FUNCTION "HMI animation unit" : VOID	// FC 60
TITLE = HMI ANIMATION FUNCTION
AUTHOR : Milesi
VERSION : 0.1
VAR_TEMP
  Temp_Start : BOOL ;
  Temp_Alm : BOOL ;
  Temp_Aux : BOOL ;
END_VAR
BEGIN
NETWORK
TITLE = LINE
      AN    "M197.0";
      =     "HMI animation".Line.DB60_DBX156_0;
NETWORK
TITLE = ALARMS PRESENT TO HMI 
      AN    "M102.1";
      O     "Db Plc <=> HMI".LINE1.DB100_DBX149_7;
      =     "HMI animation".Line.DB60_DBX156_1;
NETWORK
TITLE = LINE RUN WITH ZERO SPEED
      A     "M180.1";
      =     "HMI animation".Line.DB60_DBX156_2;
NETWORK
TITLE = PLC <--> HMI COMUNICATION CONTROL
      AN    "HMI animation".Line.DB60_DBX156_7;
      S     "HMI animation".Line.DB60_DBX156_7;
NETWORK
TITLE = TAKE-UP UNIT
// General alarm
      A(;
      ON    "M195.0";
      ON    "M195.1";
      O     "Db Plc <=> HMI".TAKE_UP_1.DB100_DBX107_2;
      );
      =     "HMI animation".Take_up_unit.DB60_DBX0_0;
// Driven pintle emergency
      A     "Db Plc <=> HMI".TRAVERSE.DB100_DBX105_0;
      =     "HMI animation".Take_up_unit.DB60_DBX0_1;
// Idle pintle emergency
      A     "Db Plc <=> HMI".TRAVERSE.DB100_DBX105_1;
      =     "HMI animation".Take_up_unit.DB60_DBX0_2;
// Bobbin up-down
      A     "MAP_DI".DB91_DBX006_0;
      A     "MAP_DI".DB91_DBX006_2;
      =     "HMI animation".Take_up_unit.DB60_DBX0_3;
// Traverse right direction
      AN    "M10.1";
      =     "HMI animation".Take_up_unit.DB60_DBX0_4;
// Traverse left direction
      A     "M10.1";
      =     "HMI animation".Take_up_unit.DB60_DBX0_5;
// Bobbin motor status
      A     "Db Plc <=> HMI".TAKE_UP_1.DB100_DBX107_4;
      O     "Db Plc <=> HMI".TAKE_UP_1.DB100_DBX107_5;
      O     "Db Plc <=> HMI".TAKE_UP_1.DB100_DBX107_6;
      =     #Temp_Aux;
      CALL  "Motor status HMI" (
           Start                    := "Plc --> Drives".BOBBIN_CONTROL_W1.DB2_DBX41_0,
           Fault                    := #Temp_Aux,
           Status_Reg               := "HMI animation".Take_up_unit.DB60_DBB1);
// Bobbin blower status
      CALL  "Motor status HMI" (
           Start                    := "MAP_DO".DB93_DBX005_1,
           Fault                    := "Db Plc <=> HMI".TAKE_UP_1.DB100_DBX107_3,
           Status_Reg               := "HMI animation".Take_up_unit.DB60_DBB2);
// Traverse motor status
      CALL  "Motor status HMI" (
           Start                    := "Plc --> Drives".TRAVERSE_CONTROL_W1.DB2_DBX1_0,
           Fault                    := "Db Plc <=> HMI".TRAVERSE.DB100_DBX105_3,
           Status_Reg               := "HMI animation".Take_up_unit.DB60_DBB3);
// Traverse blower status
      CALL  "Motor status HMI" (
           Start                    := "MAP_DO".DB93_DBX005_0,
           Fault                    := "Db Plc <=> HMI".TRAVERSE.DB100_DBX105_2,
           Status_Reg               := "HMI animation".Take_up_unit.DB60_DBB4);
// Bobbin driven pintle motor status
      A     "MAP_DO".DB93_DBX004_2;
      O     "MAP_DO".DB93_DBX004_3;
      =     #Temp_Start;
      CALL  "Motor status HMI" (
           Start                    := #Temp_Start,
           Fault                    := "Db Plc <=> HMI".TAKE_UP_1.DB100_DBX107_2,
           Status_Reg               := "HMI animation".Take_up_unit.DB60_DBB5);
// Bobbin idle pintle motor status
      A     "MAP_DO".DB93_DBX004_0;
      O     "MAP_DO".DB93_DBX004_1;
      =     #Temp_Start;
      CALL  "Motor status HMI" (
           Start                    := #Temp_Start,
           Fault                    := "Db Plc <=> HMI".TAKE_UP_1.DB100_DBX107_2,
           Status_Reg               := "HMI animation".Take_up_unit.DB60_DBB6);
// Bobbin pintle opening-closing motor status
      A     "MAP_DO".DB93_DBX004_4;
      O     "MAP_DO".DB93_DBX004_5;
      =     #Temp_Start;
      CALL  "Motor status HMI" (
           Start                    := #Temp_Start,
           Fault                    := "Db Plc <=> HMI".TAKE_UP_1.DB100_DBX107_2,
           Status_Reg               := "HMI animation".Take_up_unit.DB60_DBB7);
NETWORK
TITLE = CAPSTAN
// General alarm
      AN    "M197.3";
      =     "HMI animation".Capstan.DB60_DBX12_0;
// Cable block
      A     "MAP_DI".DB91_DBX012_3;
      =     "HMI animation".Capstan.DB60_DBX12_1;
// Motor status
      A     "Db Plc <=> HMI".CAPSTAN.DB100_DBX109_6;
      O     "Db Plc <=> HMI".CAPSTAN.DB100_DBX109_7;
      =     #Temp_Alm;
      CALL  "Motor status HMI" (
           Start                    := "Plc --> Drives".CAPSTAN_CONTROL_W1.DB2_DBX81_0,
           Fault                    := #Temp_Alm,
           Status_Reg               := "HMI animation".Capstan.DB60_DBB13);
// Blower status
      CALL  "Motor status HMI" (
           Start                    := "MAP_DO".DB93_DBX001_2,
           Fault                    := "Db Plc <=> HMI".CAPSTAN.DB100_DBX109_0,
           Status_Reg               := "HMI animation".Capstan.DB60_DBB14);
NETWORK
TITLE = CAGE 24
// General alarm
      AN    "M195.3";
      O     "Db Plc <=> HMI".CAGE24_1.DB100_DBX112_02;
      O     "Db Plc <=> HMI".CAGE24_1.DB100_DBX112_04;
      O     "Db Plc <=> HMI".CAGE24_1.DB100_DBX113_05;
      =     "HMI animation".Cage_24.DB60_DBX36_0;
// Motor status
      A     "Db Plc <=> HMI".CAGE24_4.DB100_DBX118_05;
      O     "Db Plc <=> HMI".CAGE24_4.DB100_DBX118_06;
      =     #Temp_Alm;
      CALL  "Motor status HMI" (
           Start                    := "Plc --> Drives".CAGE_24_CONTROL_W1.DB2_DBX161_0,
           Fault                    := #Temp_Alm,
           Status_Reg               := "HMI animation".Cage_24.DB60_DBB37);
// Blower status
      CALL  "Motor status HMI" (
           Start                    := "MAP_DO".DB93_DBX018_2,
           Fault                    := "Db Plc <=> HMI".CAGE24_1.DB100_DBX113_02,
           Status_Reg               := "HMI animation".Cage_24.DB60_DBB38);
// Loading motor status
      A     "MAP_DO".DB93_DBX018_4;
      O     "MAP_DO".DB93_DBX018_3;
      =     #Temp_Start;
      CALL  "Motor status HMI" (
           Start                    := #Temp_Start,
           Fault                    := "Db Plc <=> HMI".CAGE24_1.DB100_DBX112_04,
           Status_Reg               := "HMI animation".Cage_24.DB60_DBB39);
NETWORK
TITLE = CAGE 24 PREFORMING
// General alarm
      AN    "M195.4";
      =     "HMI animation".Cage_24_preforming.DB60_DBX48_0;
// Motor status
      A     "Db Plc <=> HMI".CAGE24_4.DB100_DBX119_04;
      O     "Db Plc <=> HMI".CAGE24_4.DB100_DBX119_07;
      =     #Temp_Alm;
      CALL  "Motor status HMI" (
           Start                    := "Plc --> Drives".CAGE_24_PREF_CONTROL_W1.DB2_DBX121_0,
           Fault                    := #Temp_Alm,
           Status_Reg               := "HMI animation".Cage_24_preforming.DB60_DBB49);
// Blower status
      CALL  "Motor status HMI" (
           Start                    := "MAP_DO".DB93_DBX018_1,
           Fault                    := "Db Plc <=> HMI".CAGE24_4.DB100_DBX119_05,
           Status_Reg               := "HMI animation".Cage_24_preforming.DB60_DBB50);
NETWORK
TITLE = CAGE 18
// General alarm
      AN    "M195.5";
      O     "Db Plc <=> HMI".CAGE18_1.DB100_DBX120_02;
      O     "Db Plc <=> HMI".CAGE18_1.DB100_DBX120_04;
      O     "Db Plc <=> HMI".CAGE18_1.DB100_DBX121_05;
      =     "HMI animation".Cage_18.DB60_DBX60_0;
// Motor status
      A     "Db Plc <=> HMI".CAGE18_4.DB100_DBX126_05;
      O     "Db Plc <=> HMI".CAGE18_4.DB100_DBX126_06;
      =     #Temp_Alm;
      CALL  "Motor status HMI" (
           Start                    := "Plc --> Drives".CAGE_18_CONTROL_W1.DB2_DBX241_0,
           Fault                    := #Temp_Alm,
           Status_Reg               := "HMI animation".Cage_18.DB60_DBB61);
// Blower status
      CALL  "Motor status HMI" (
           Start                    := "MAP_DO".DB93_DBX028_2,
           Fault                    := "Db Plc <=> HMI".CAGE18_1.DB100_DBX121_02,
           Status_Reg               := "HMI animation".Cage_18.DB60_DBB62);
// Loading motor status
      A     "MAP_DO".DB93_DBX028_4;
      O     "MAP_DO".DB93_DBX028_3;
      =     #Temp_Start;
      CALL  "Motor status HMI" (
           Start                    := #Temp_Start,
           Fault                    := "Db Plc <=> HMI".CAGE18_1.DB100_DBX120_04,
           Status_Reg               := "HMI animation".Cage_18.DB60_DBB63);
NETWORK
TITLE = CAGE 18 PREFORMING
// General alarm
      AN    "M195.6";
      =     "HMI animation".Cage_18_preforming.DB60_DBX72_0;
// Motor status
      A     "Db Plc <=> HMI".CAGE18_4.DB100_DBX127_04;
      O     "Db Plc <=> HMI".CAGE18_4.DB100_DBX127_07;
      =     #Temp_Alm;
      CALL  "Motor status HMI" (
           Start                    := "Plc --> Drives".CAGE_18_PREF_CONTROL_W1.DB2_DBX201_0,
           Fault                    := #Temp_Alm,
           Status_Reg               := "HMI animation".Cage_18_preforming.DB60_DBB73);
// Blower status
      CALL  "Motor status HMI" (
           Start                    := "MAP_DO".DB93_DBX028_1,
           Fault                    := "Db Plc <=> HMI".CAGE18_4.DB100_DBX127_05,
           Status_Reg               := "HMI animation".Cage_18_preforming.DB60_DBB74);
NETWORK
TITLE = CAGE 12
// General alarm
      AN    "M195.7";
      O     "Db Plc <=> HMI".CAGE12_1.DB100_DBX128_02;
      O     "Db Plc <=> HMI".CAGE12_1.DB100_DBX128_06;
      O     "Db Plc <=> HMI".CAGE12_1.DB100_DBX129_05;
      =     "HMI animation".Cage_12.DB60_DBX84_0;
// Motor status
      A     "Db Plc <=> HMI".Cage12_4.DB100_DBX134_05;
      O     "Db Plc <=> HMI".Cage12_4.DB100_DBX134_06;
      =     #Temp_Alm;
      CALL  "Motor status HMI" (
           Start                    := "Plc --> Drives".CAGE_12_CONTROL_W1.DB2_DBX321_0,
           Fault                    := #Temp_Alm,
           Status_Reg               := "HMI animation".Cage_12.DB60_DBB85);
// Blower status
      CALL  "Motor status HMI" (
           Start                    := "MAP_DO".DB93_DBX038_2,
           Fault                    := "Db Plc <=> HMI".CAGE12_1.DB100_DBX129_02,
           Status_Reg               := "HMI animation".Cage_12.DB60_DBB86);
// Loading motor status
      A     "MAP_DO".DB93_DBX038_4;
      O     "MAP_DO".DB93_DBX038_3;
      =     #Temp_Start;
      CALL  "Motor status HMI" (
           Start                    := #Temp_Start,
           Fault                    := "Db Plc <=> HMI".CAGE12_1.DB100_DBX128_06,
           Status_Reg               := "HMI animation".Cage_12.DB60_DBB87);
NETWORK
TITLE = CAGE 12 PREFORMING
// General alarm
      AN    "M196.0";
      =     "HMI animation".Cage_12_preforming.DB60_DBX96_0;
// Motor status
      A     "Db Plc <=> HMI".Cage12_4.DB100_DBX135_04;
      O     "Db Plc <=> HMI".Cage12_4.DB100_DBX135_07;
      =     #Temp_Alm;
      CALL  "Motor status HMI" (
           Start                    := "Plc --> Drives".CAGE_12_PREF_CONTROL_W1.DB2_DBX281_0,
           Fault                    := #Temp_Alm,
           Status_Reg               := "HMI animation".Cage_12_preforming.DB60_DBB97);
// Blower status
      CALL  "Motor status HMI" (
           Start                    := "MAP_DO".DB93_DBX038_1,
           Fault                    := "Db Plc <=> HMI".Cage12_4.DB100_DBX135_05,
           Status_Reg               := "HMI animation".Cage_12_preforming.DB60_DBB98);
NETWORK
TITLE = CAGE 6
// General alarm
      AN    "M196.1";
      O     "Db Plc <=> HMI".Cage6_1.DB100_DBX136_2;
      O     "Db Plc <=> HMI".Cage6_1.DB100_DBX136_6;
      O     "Db Plc <=> HMI".Cage6_1.DB100_DBX137_5;
      =     "HMI animation".Cage_6.DB60_DBX108_0;
// Motor status
      A     "Db Plc <=> HMI".Cage6_4.DB100_DBX142_5;
      O     "Db Plc <=> HMI".Cage6_4.DB100_DBX142_6;
      =     #Temp_Alm;
      CALL  "Motor status HMI" (
           Start                    := "Plc --> Drives".CAGE_6_CONTROL_W1.DB2_DBX361_0,
           Fault                    := #Temp_Alm,
           Status_Reg               := "HMI animation".Cage_6.DB60_DBB109);
// Blower status
      CALL  "Motor status HMI" (
           Start                    := "MAP_DO".DB93_DBX048_2,
           Fault                    := "Db Plc <=> HMI".Cage6_1.DB100_DBX137_2,
           Status_Reg               := "HMI animation".Cage_6.DB60_DBB110);
// Loading motor status
      A     "MAP_DO".DB93_DBX048_3;
      O     "MAP_DO".DB93_DBX048_4;
      =     #Temp_Start;
      CALL  "Motor status HMI" (
           Start                    := #Temp_Start,
           Fault                    := "Db Plc <=> HMI".Cage6_1.DB100_DBX136_6,
           Status_Reg               := "HMI animation".Cage_6.DB60_DBB111);
NETWORK
TITLE = CAGE 6 PREFORMING
// General alarm
      AN    "M196.2";
      =     "HMI animation".Cage_6_preforming.DB60_DBX120_0;
NETWORK
TITLE = PAY-OFF 630 UNIT
// General alarm
      AN    "M196.3";
      =     "HMI animation".Pay_off_630.DB60_DBX132_0;
      A     "MAP_DI".DB91_DBX099_0;
      =     "HMI animation".Pay_off_630.DB60_DBX132_1;
END_FUNCTION

FUNCTION "Take-up traverse impulse" : VOID	// FC 61
TITLE = TAKE-UP TRAVERSE IMPULSES FUNCTION
AUTHOR : Milesi
VERSION : 0.1
VAR_TEMP
  Traverse_Encoder_Caunt : DINT ;
END_VAR
BEGIN
NETWORK
TITLE = COUNT 24V/100kHz SETTINGS
//Presettings
      L     0;
      T     "Count setting".DINT0;
      T     "Count setting".DINT4;
      SET;
      S     DB101.DBX 4.0;
//Command interface writing
      L     "Count setting".DINT0;
      T     "PAD272";
      L     DB101.DBW 4;
      T     "PAW276";
//Status interface reading
      L     "PED272";
      T     "Count setting".DINT8;
      L     "PED276";
      T     "Count setting".DINT12;
NETWORK
TITLE = TAKE-UP TRAVERSE ENCODER COUNT
      L     "Count setting".DINT8;
      NEGD;
      T     #Traverse_Encoder_Caunt;
NETWORK
TITLE = TAKE-UP TRAVERSE POSITION QUOTA CALCULATION
      L     #Traverse_Encoder_Caunt;
      L     "Take-up traverse".DB5_DBD44;
      -D;
      DTR;
      L     1.793919e-03;
      *R;
      T     "Take-up traverse".DB5_DBD40;
      L     #Traverse_Encoder_Caunt;
      T     "Take-up traverse".DB5_DBD44;
NETWORK
TITLE = TRAVERSE QUOTA INCREASE
      L     "Take-up traverse".DB5_DBD40;
      L     "Take-up traverse".DB5_DBD32;
      +R;
      T     "Take-up traverse".DB5_DBD32;
NETWORK
TITLE = TAKE-UP TRAVERSE POSITION QUOTA RESET
      A     "MAP_DI".DB91_DBX008_4;
      JNB   _023;
      L     0.000000e+00;
      T     "Take-up traverse".DB5_DBD32;
_023: NOP   0;
END_FUNCTION

FUNCTION "Cage 24 wires insertion" : VOID	// FC 70
TITLE = CAGE 24 WIRES INSERTION AND ALARM FUNCTION
AUTHOR : Milesi
VERSION : 0.1
VAR_TEMP
  Tres : BOOL ;
END_VAR
BEGIN
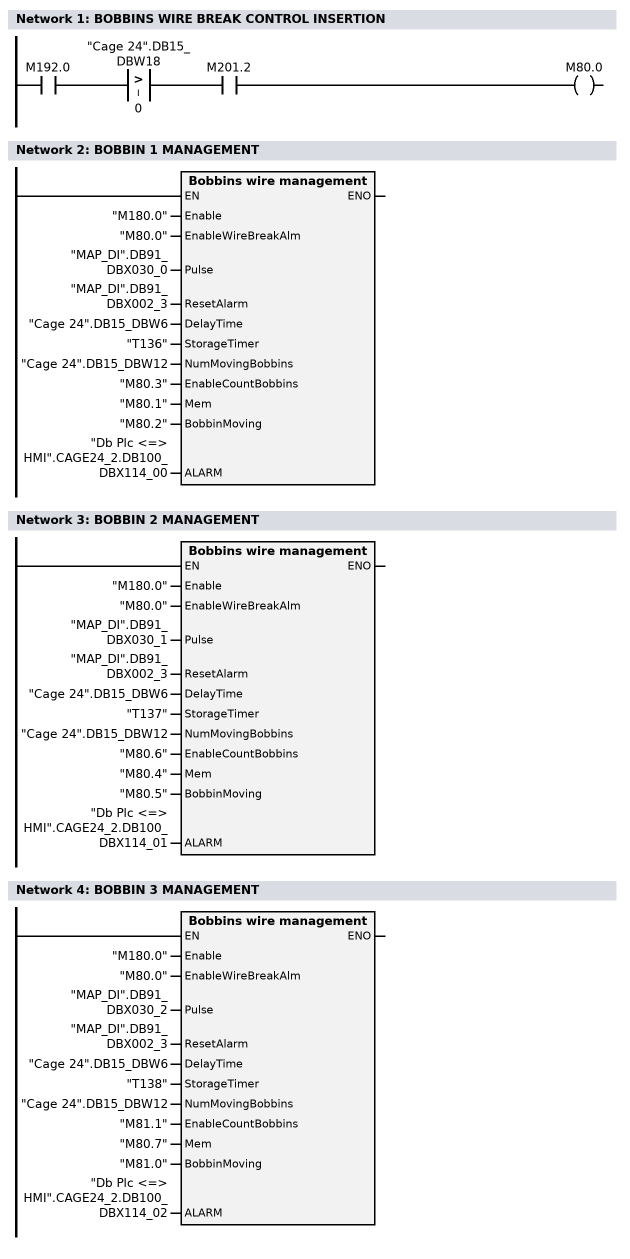
NETWORK
TITLE = BOBBINS WIRE BREAK CONTROL INSERTION
      A     "M192.0";
      A(;
      L     "Cage 24".DB15_DBW18;
      L     0;
      >I;
      );
      A     "M201.2";
      =     "M80.0";
NETWORK
TITLE = BOBBIN 1 MANAGEMENT
      CALL  "Bobbins wire management" (
           Enable                   := "M180.0",
           EnableWireBreakAlm       := "M80.0",
           Pulse                    := "MAP_DI".DB91_DBX030_0,
           ResetAlarm               := "MAP_DI".DB91_DBX002_3,
           DelayTime                := "Cage 24".DB15_DBW6,
           StorageTimer             := "T136",
           NumMovingBobbins         := "Cage 24".DB15_DBW12,
           EnableCountBobbins       := "M80.3",
           Mem                      := "M80.1",
           BobbinMoving             := "M80.2",
           ALARM                    := "Db Plc <=> HMI".CAGE24_2.DB100_DBX114_00);
      NOP   0;
NETWORK
TITLE = BOBBIN 2 MANAGEMENT
      CALL  "Bobbins wire management" (
           Enable                   := "M180.0",
           EnableWireBreakAlm       := "M80.0",
           Pulse                    := "MAP_DI".DB91_DBX030_1,
           ResetAlarm               := "MAP_DI".DB91_DBX002_3,
           DelayTime                := "Cage 24".DB15_DBW6,
           StorageTimer             := "T137",
           NumMovingBobbins         := "Cage 24".DB15_DBW12,
           EnableCountBobbins       := "M80.6",
           Mem                      := "M80.4",
           BobbinMoving             := "M80.5",
           ALARM                    := "Db Plc <=> HMI".CAGE24_2.DB100_DBX114_01);
NETWORK
TITLE = BOBBIN 3 MANAGEMENT
      CALL  "Bobbins wire management" (
           Enable                   := "M180.0",
           EnableWireBreakAlm       := "M80.0",
           Pulse                    := "MAP_DI".DB91_DBX030_2,
           ResetAlarm               := "MAP_DI".DB91_DBX002_3,
           DelayTime                := "Cage 24".DB15_DBW6,
           StorageTimer             := "T138",
           NumMovingBobbins         := "Cage 24".DB15_DBW12,
           EnableCountBobbins       := "M81.1",
           Mem                      := "M80.7",
           BobbinMoving             := "M81.0",
           ALARM                    := "Db Plc <=> HMI".CAGE24_2.DB100_DBX114_02);
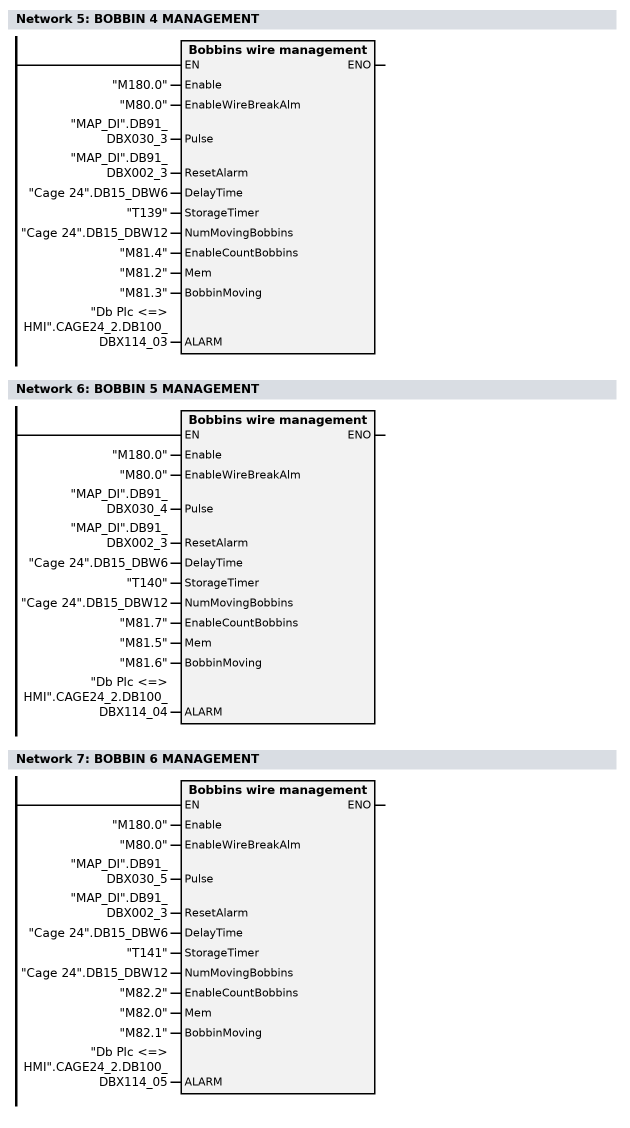
NETWORK
TITLE = BOBBIN 4 MANAGEMENT
      CALL  "Bobbins wire management" (
           Enable                   := "M180.0",
           EnableWireBreakAlm       := "M80.0",
           Pulse                    := "MAP_DI".DB91_DBX030_3,
           ResetAlarm               := "MAP_DI".DB91_DBX002_3,
           DelayTime                := "Cage 24".DB15_DBW6,
           StorageTimer             := "T139",
           NumMovingBobbins         := "Cage 24".DB15_DBW12,
           EnableCountBobbins       := "M81.4",
           Mem                      := "M81.2",
           BobbinMoving             := "M81.3",
           ALARM                    := "Db Plc <=> HMI".CAGE24_2.DB100_DBX114_03);
NETWORK
TITLE = BOBBIN 5 MANAGEMENT
      CALL  "Bobbins wire management" (
           Enable                   := "M180.0",
           EnableWireBreakAlm       := "M80.0",
           Pulse                    := "MAP_DI".DB91_DBX030_4,
           ResetAlarm               := "MAP_DI".DB91_DBX002_3,
           DelayTime                := "Cage 24".DB15_DBW6,
           StorageTimer             := "T140",
           NumMovingBobbins         := "Cage 24".DB15_DBW12,
           EnableCountBobbins       := "M81.7",
           Mem                      := "M81.5",
           BobbinMoving             := "M81.6",
           ALARM                    := "Db Plc <=> HMI".CAGE24_2.DB100_DBX114_04);
NETWORK
TITLE = BOBBIN 6 MANAGEMENT
      CALL  "Bobbins wire management" (
           Enable                   := "M180.0",
           EnableWireBreakAlm       := "M80.0",
           Pulse                    := "MAP_DI".DB91_DBX030_5,
           ResetAlarm               := "MAP_DI".DB91_DBX002_3,
           DelayTime                := "Cage 24".DB15_DBW6,
           StorageTimer             := "T141",
           NumMovingBobbins         := "Cage 24".DB15_DBW12,
           EnableCountBobbins       := "M82.2",
           Mem                      := "M82.0",
           BobbinMoving             := "M82.1",
           ALARM                    := "Db Plc <=> HMI".CAGE24_2.DB100_DBX114_05);
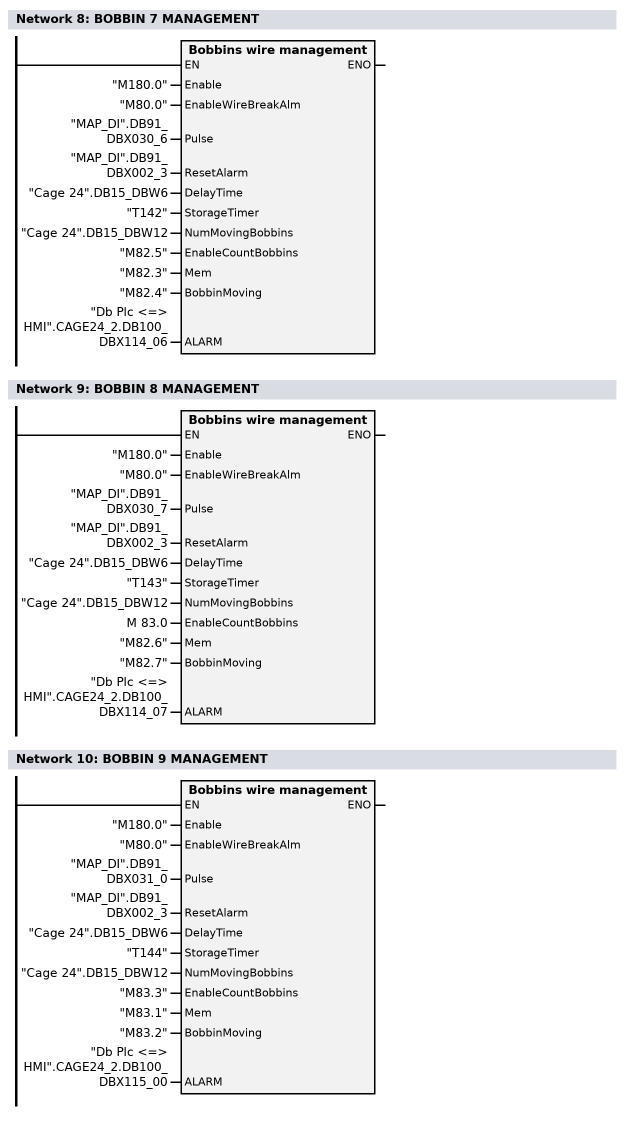
NETWORK
TITLE = BOBBIN 7 MANAGEMENT
      CALL  "Bobbins wire management" (
           Enable                   := "M180.0",
           EnableWireBreakAlm       := "M80.0",
           Pulse                    := "MAP_DI".DB91_DBX030_6,
           ResetAlarm               := "MAP_DI".DB91_DBX002_3,
           DelayTime                := "Cage 24".DB15_DBW6,
           StorageTimer             := "T142",
           NumMovingBobbins         := "Cage 24".DB15_DBW12,
           EnableCountBobbins       := "M82.5",
           Mem                      := "M82.3",
           BobbinMoving             := "M82.4",
           ALARM                    := "Db Plc <=> HMI".CAGE24_2.DB100_DBX114_06);
NETWORK
TITLE = BOBBIN 8 MANAGEMENT
      CALL  "Bobbins wire management" (
           Enable                   := "M180.0",
           EnableWireBreakAlm       := "M80.0",
           Pulse                    := "MAP_DI".DB91_DBX030_7,
           ResetAlarm               := "MAP_DI".DB91_DBX002_3,
           DelayTime                := "Cage 24".DB15_DBW6,
           StorageTimer             := "T143",
           NumMovingBobbins         := "Cage 24".DB15_DBW12,
           EnableCountBobbins       := M 83.0,
           Mem                      := "M82.6",
           BobbinMoving             := "M82.7",
           ALARM                    := "Db Plc <=> HMI".CAGE24_2.DB100_DBX114_07);
NETWORK
TITLE = BOBBIN 9 MANAGEMENT
      CALL  "Bobbins wire management" (
           Enable                   := "M180.0",
           EnableWireBreakAlm       := "M80.0",
           Pulse                    := "MAP_DI".DB91_DBX031_0,
           ResetAlarm               := "MAP_DI".DB91_DBX002_3,
           DelayTime                := "Cage 24".DB15_DBW6,
           StorageTimer             := "T144",
           NumMovingBobbins         := "Cage 24".DB15_DBW12,
           EnableCountBobbins       := "M83.3",
           Mem                      := "M83.1",
           BobbinMoving             := "M83.2",
           ALARM                    := "Db Plc <=> HMI".CAGE24_2.DB100_DBX115_00);
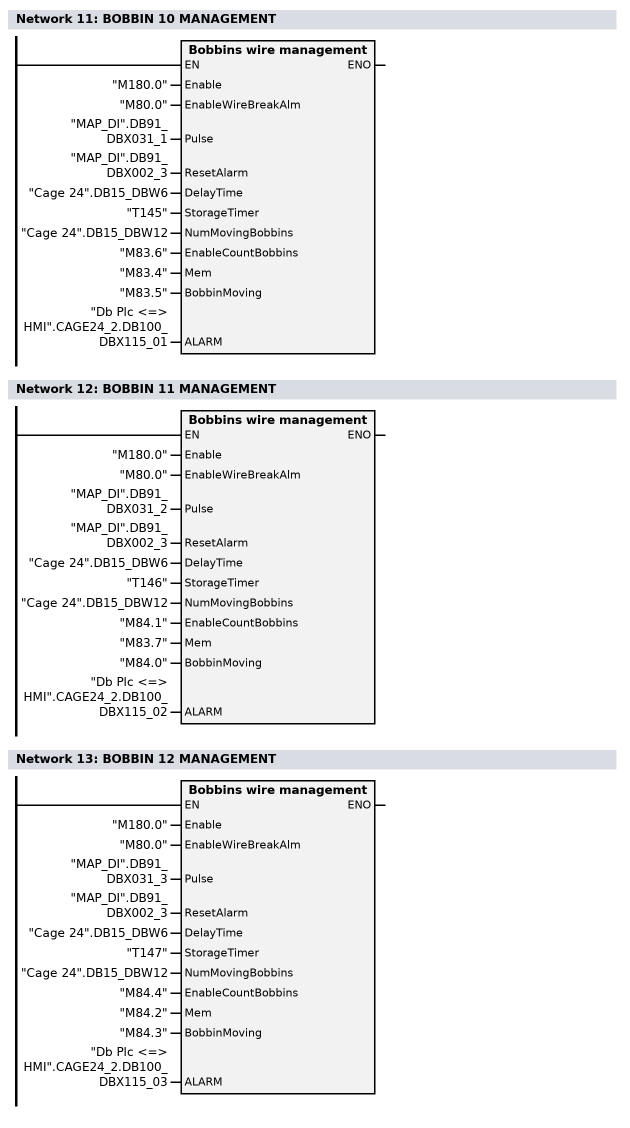
NETWORK
TITLE = BOBBIN 10 MANAGEMENT
      CALL  "Bobbins wire management" (
           Enable                   := "M180.0",
           EnableWireBreakAlm       := "M80.0",
           Pulse                    := "MAP_DI".DB91_DBX031_1,
           ResetAlarm               := "MAP_DI".DB91_DBX002_3,
           DelayTime                := "Cage 24".DB15_DBW6,
           StorageTimer             := "T145",
           NumMovingBobbins         := "Cage 24".DB15_DBW12,
           EnableCountBobbins       := "M83.6",
           Mem                      := "M83.4",
           BobbinMoving             := "M83.5",
           ALARM                    := "Db Plc <=> HMI".CAGE24_2.DB100_DBX115_01);
NETWORK
TITLE = BOBBIN 11 MANAGEMENT
      CALL  "Bobbins wire management" (
           Enable                   := "M180.0",
           EnableWireBreakAlm       := "M80.0",
           Pulse                    := "MAP_DI".DB91_DBX031_2,
           ResetAlarm               := "MAP_DI".DB91_DBX002_3,
           DelayTime                := "Cage 24".DB15_DBW6,
           StorageTimer             := "T146",
           NumMovingBobbins         := "Cage 24".DB15_DBW12,
           EnableCountBobbins       := "M84.1",
           Mem                      := "M83.7",
           BobbinMoving             := "M84.0",
           ALARM                    := "Db Plc <=> HMI".CAGE24_2.DB100_DBX115_02);
NETWORK
TITLE = BOBBIN 12 MANAGEMENT
      CALL  "Bobbins wire management" (
           Enable                   := "M180.0",
           EnableWireBreakAlm       := "M80.0",
           Pulse                    := "MAP_DI".DB91_DBX031_3,
           ResetAlarm               := "MAP_DI".DB91_DBX002_3,
           DelayTime                := "Cage 24".DB15_DBW6,
           StorageTimer             := "T147",
           NumMovingBobbins         := "Cage 24".DB15_DBW12,
           EnableCountBobbins       := "M84.4",
           Mem                      := "M84.2",
           BobbinMoving             := "M84.3",
           ALARM                    := "Db Plc <=> HMI".CAGE24_2.DB100_DBX115_03);
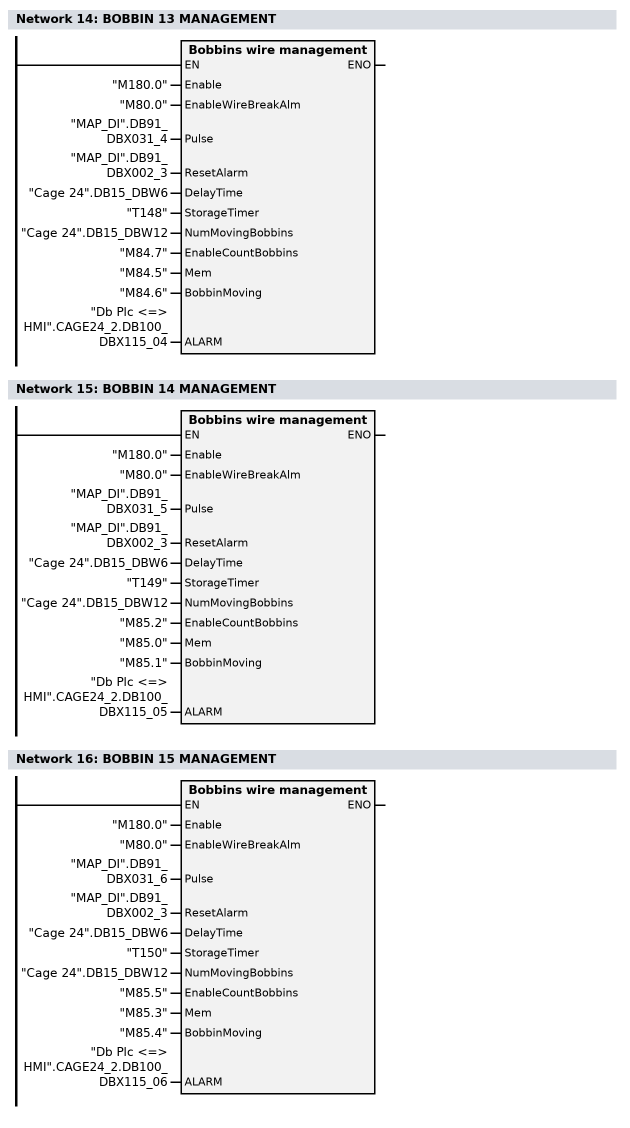
NETWORK
TITLE = BOBBIN 13 MANAGEMENT
      CALL  "Bobbins wire management" (
           Enable                   := "M180.0",
           EnableWireBreakAlm       := "M80.0",
           Pulse                    := "MAP_DI".DB91_DBX031_4,
           ResetAlarm               := "MAP_DI".DB91_DBX002_3,
           DelayTime                := "Cage 24".DB15_DBW6,
           StorageTimer             := "T148",
           NumMovingBobbins         := "Cage 24".DB15_DBW12,
           EnableCountBobbins       := "M84.7",
           Mem                      := "M84.5",
           BobbinMoving             := "M84.6",
           ALARM                    := "Db Plc <=> HMI".CAGE24_2.DB100_DBX115_04);
NETWORK
TITLE = BOBBIN 14 MANAGEMENT
      CALL  "Bobbins wire management" (
           Enable                   := "M180.0",
           EnableWireBreakAlm       := "M80.0",
           Pulse                    := "MAP_DI".DB91_DBX031_5,
           ResetAlarm               := "MAP_DI".DB91_DBX002_3,
           DelayTime                := "Cage 24".DB15_DBW6,
           StorageTimer             := "T149",
           NumMovingBobbins         := "Cage 24".DB15_DBW12,
           EnableCountBobbins       := "M85.2",
           Mem                      := "M85.0",
           BobbinMoving             := "M85.1",
           ALARM                    := "Db Plc <=> HMI".CAGE24_2.DB100_DBX115_05);
NETWORK
TITLE = BOBBIN 15 MANAGEMENT
      CALL  "Bobbins wire management" (
           Enable                   := "M180.0",
           EnableWireBreakAlm       := "M80.0",
           Pulse                    := "MAP_DI".DB91_DBX031_6,
           ResetAlarm               := "MAP_DI".DB91_DBX002_3,
           DelayTime                := "Cage 24".DB15_DBW6,
           StorageTimer             := "T150",
           NumMovingBobbins         := "Cage 24".DB15_DBW12,
           EnableCountBobbins       := "M85.5",
           Mem                      := "M85.3",
           BobbinMoving             := "M85.4",
           ALARM                    := "Db Plc <=> HMI".CAGE24_2.DB100_DBX115_06);
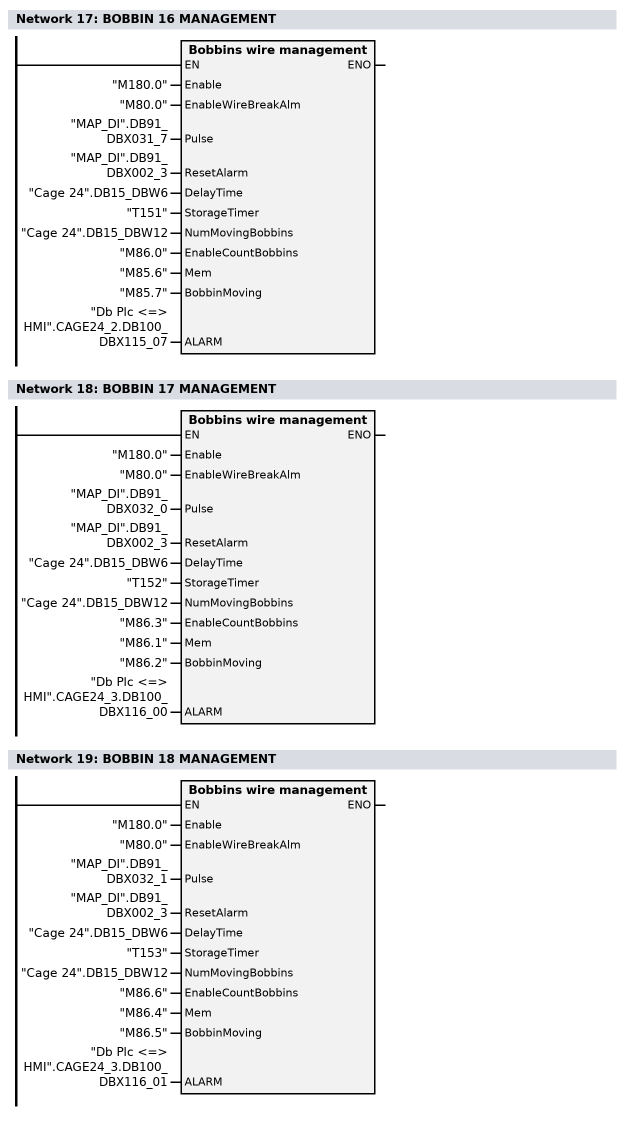
NETWORK
TITLE = BOBBIN 16 MANAGEMENT
      CALL  "Bobbins wire management" (
           Enable                   := "M180.0",
           EnableWireBreakAlm       := "M80.0",
           Pulse                    := "MAP_DI".DB91_DBX031_7,
           ResetAlarm               := "MAP_DI".DB91_DBX002_3,
           DelayTime                := "Cage 24".DB15_DBW6,
           StorageTimer             := "T151",
           NumMovingBobbins         := "Cage 24".DB15_DBW12,
           EnableCountBobbins       := "M86.0",
           Mem                      := "M85.6",
           BobbinMoving             := "M85.7",
           ALARM                    := "Db Plc <=> HMI".CAGE24_2.DB100_DBX115_07);
NETWORK
TITLE = BOBBIN 17 MANAGEMENT
      CALL  "Bobbins wire management" (
           Enable                   := "M180.0",
           EnableWireBreakAlm       := "M80.0",
           Pulse                    := "MAP_DI".DB91_DBX032_0,
           ResetAlarm               := "MAP_DI".DB91_DBX002_3,
           DelayTime                := "Cage 24".DB15_DBW6,
           StorageTimer             := "T152",
           NumMovingBobbins         := "Cage 24".DB15_DBW12,
           EnableCountBobbins       := "M86.3",
           Mem                      := "M86.1",
           BobbinMoving             := "M86.2",
           ALARM                    := "Db Plc <=> HMI".CAGE24_3.DB100_DBX116_00);
NETWORK
TITLE = BOBBIN 18 MANAGEMENT
      CALL  "Bobbins wire management" (
           Enable                   := "M180.0",
           EnableWireBreakAlm       := "M80.0",
           Pulse                    := "MAP_DI".DB91_DBX032_1,
           ResetAlarm               := "MAP_DI".DB91_DBX002_3,
           DelayTime                := "Cage 24".DB15_DBW6,
           StorageTimer             := "T153",
           NumMovingBobbins         := "Cage 24".DB15_DBW12,
           EnableCountBobbins       := "M86.6",
           Mem                      := "M86.4",
           BobbinMoving             := "M86.5",
           ALARM                    := "Db Plc <=> HMI".CAGE24_3.DB100_DBX116_01);
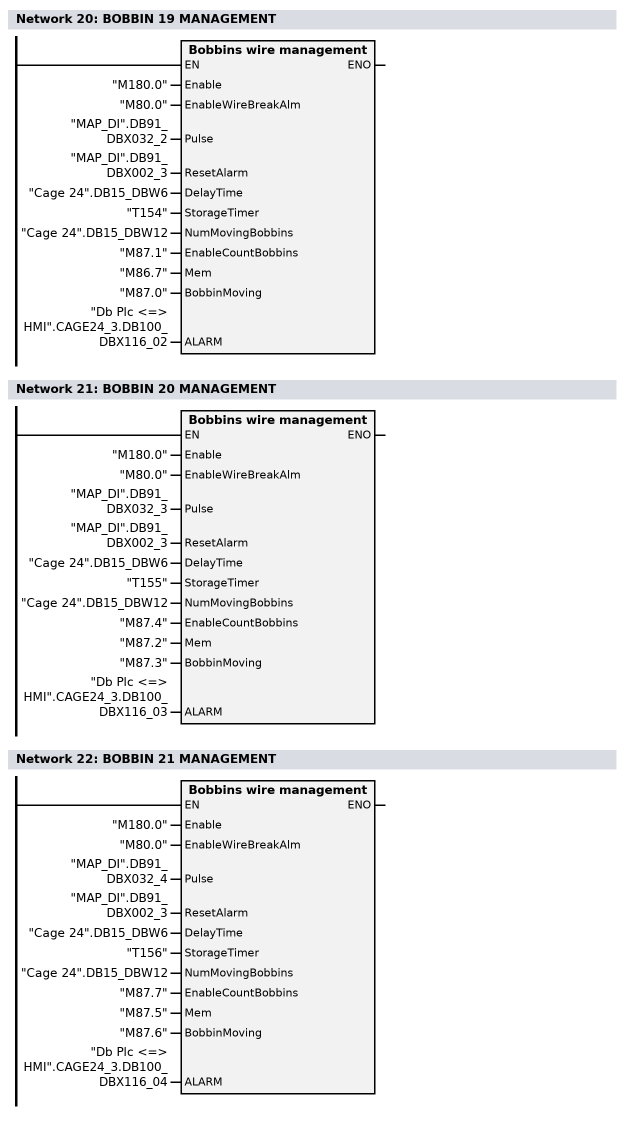
NETWORK
TITLE = BOBBIN 19 MANAGEMENT
      CALL  "Bobbins wire management" (
           Enable                   := "M180.0",
           EnableWireBreakAlm       := "M80.0",
           Pulse                    := "MAP_DI".DB91_DBX032_2,
           ResetAlarm               := "MAP_DI".DB91_DBX002_3,
           DelayTime                := "Cage 24".DB15_DBW6,
           StorageTimer             := "T154",
           NumMovingBobbins         := "Cage 24".DB15_DBW12,
           EnableCountBobbins       := "M87.1",
           Mem                      := "M86.7",
           BobbinMoving             := "M87.0",
           ALARM                    := "Db Plc <=> HMI".CAGE24_3.DB100_DBX116_02);
NETWORK
TITLE = BOBBIN 20 MANAGEMENT
      CALL  "Bobbins wire management" (
           Enable                   := "M180.0",
           EnableWireBreakAlm       := "M80.0",
           Pulse                    := "MAP_DI".DB91_DBX032_3,
           ResetAlarm               := "MAP_DI".DB91_DBX002_3,
           DelayTime                := "Cage 24".DB15_DBW6,
           StorageTimer             := "T155",
           NumMovingBobbins         := "Cage 24".DB15_DBW12,
           EnableCountBobbins       := "M87.4",
           Mem                      := "M87.2",
           BobbinMoving             := "M87.3",
           ALARM                    := "Db Plc <=> HMI".CAGE24_3.DB100_DBX116_03);
NETWORK
TITLE = BOBBIN 21 MANAGEMENT
      CALL  "Bobbins wire management" (
           Enable                   := "M180.0",
           EnableWireBreakAlm       := "M80.0",
           Pulse                    := "MAP_DI".DB91_DBX032_4,
           ResetAlarm               := "MAP_DI".DB91_DBX002_3,
           DelayTime                := "Cage 24".DB15_DBW6,
           StorageTimer             := "T156",
           NumMovingBobbins         := "Cage 24".DB15_DBW12,
           EnableCountBobbins       := "M87.7",
           Mem                      := "M87.5",
           BobbinMoving             := "M87.6",
           ALARM                    := "Db Plc <=> HMI".CAGE24_3.DB100_DBX116_04);
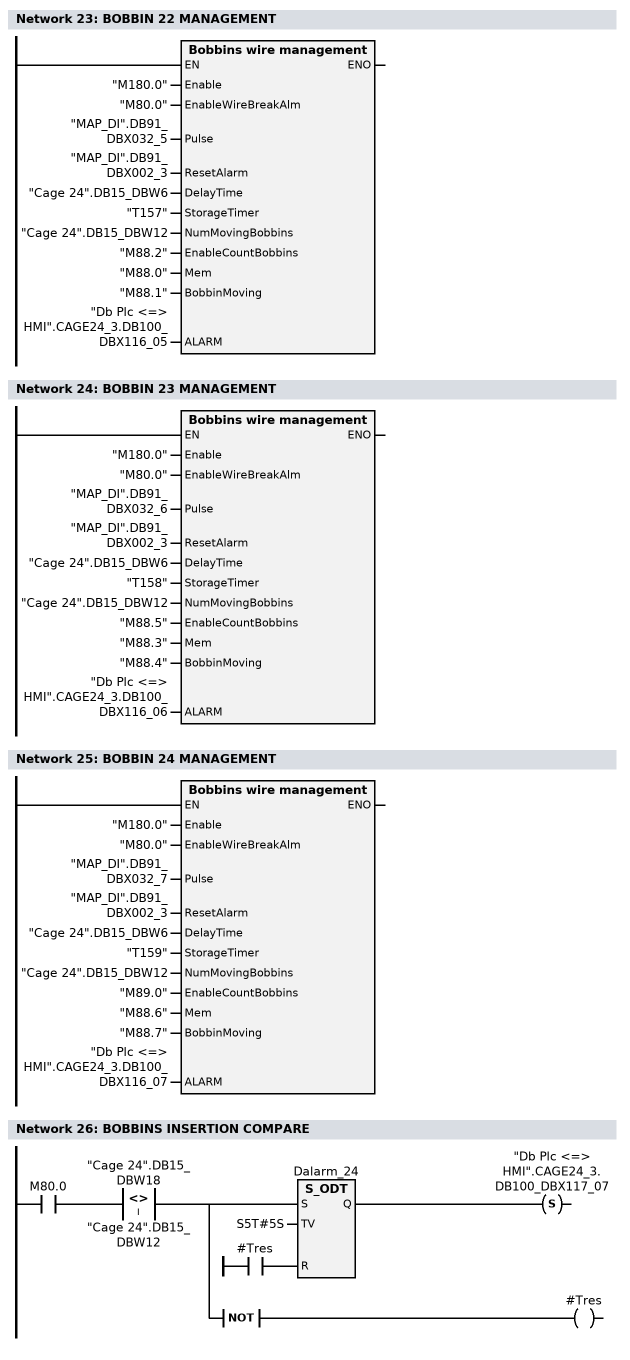
NETWORK
TITLE = BOBBIN 22 MANAGEMENT
      CALL  "Bobbins wire management" (
           Enable                   := "M180.0",
           EnableWireBreakAlm       := "M80.0",
           Pulse                    := "MAP_DI".DB91_DBX032_5,
           ResetAlarm               := "MAP_DI".DB91_DBX002_3,
           DelayTime                := "Cage 24".DB15_DBW6,
           StorageTimer             := "T157",
           NumMovingBobbins         := "Cage 24".DB15_DBW12,
           EnableCountBobbins       := "M88.2",
           Mem                      := "M88.0",
           BobbinMoving             := "M88.1",
           ALARM                    := "Db Plc <=> HMI".CAGE24_3.DB100_DBX116_05);
NETWORK
TITLE = BOBBIN 23 MANAGEMENT
      CALL  "Bobbins wire management" (
           Enable                   := "M180.0",
           EnableWireBreakAlm       := "M80.0",
           Pulse                    := "MAP_DI".DB91_DBX032_6,
           ResetAlarm               := "MAP_DI".DB91_DBX002_3,
           DelayTime                := "Cage 24".DB15_DBW6,
           StorageTimer             := "T158",
           NumMovingBobbins         := "Cage 24".DB15_DBW12,
           EnableCountBobbins       := "M88.5",
           Mem                      := "M88.3",
           BobbinMoving             := "M88.4",
           ALARM                    := "Db Plc <=> HMI".CAGE24_3.DB100_DBX116_06);
NETWORK
TITLE = BOBBIN 24 MANAGEMENT
      CALL  "Bobbins wire management" (
           Enable                   := "M180.0",
           EnableWireBreakAlm       := "M80.0",
           Pulse                    := "MAP_DI".DB91_DBX032_7,
           ResetAlarm               := "MAP_DI".DB91_DBX002_3,
           DelayTime                := "Cage 24".DB15_DBW6,
           StorageTimer             := "T159",
           NumMovingBobbins         := "Cage 24".DB15_DBW12,
           EnableCountBobbins       := "M89.0",
           Mem                      := "M88.6",
           BobbinMoving             := "M88.7",
           ALARM                    := "Db Plc <=> HMI".CAGE24_3.DB100_DBX116_07);
NETWORK
TITLE = BOBBINS INSERTION COMPARE
      A     "M80.0";
      A(;
      L     "Cage 24".DB15_DBW18;
      L     "Cage 24".DB15_DBW12;
      <>I;
      );
      =     L 1.0;
      A     L 1.0;
      L     S5T#5S;
      SD    "Dalarm_24";
      A     #Tres;
      R     "Dalarm_24";
      NOP   0;
      NOP   0;
      A     "Dalarm_24";
      S     "Db Plc <=> HMI".CAGE24_3.DB100_DBX117_07;
      A     L 1.0;
      NOT;
      =     #Tres;
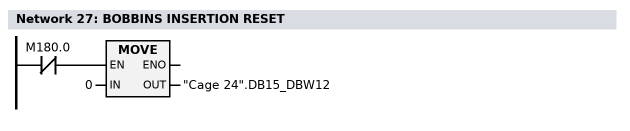
NETWORK
TITLE = BOBBINS INSERTION RESET
      AN    "M180.0";
      JNB   _001;
      L     0;
      T     "Cage 24".DB15_DBW12;
_001: NOP   0;
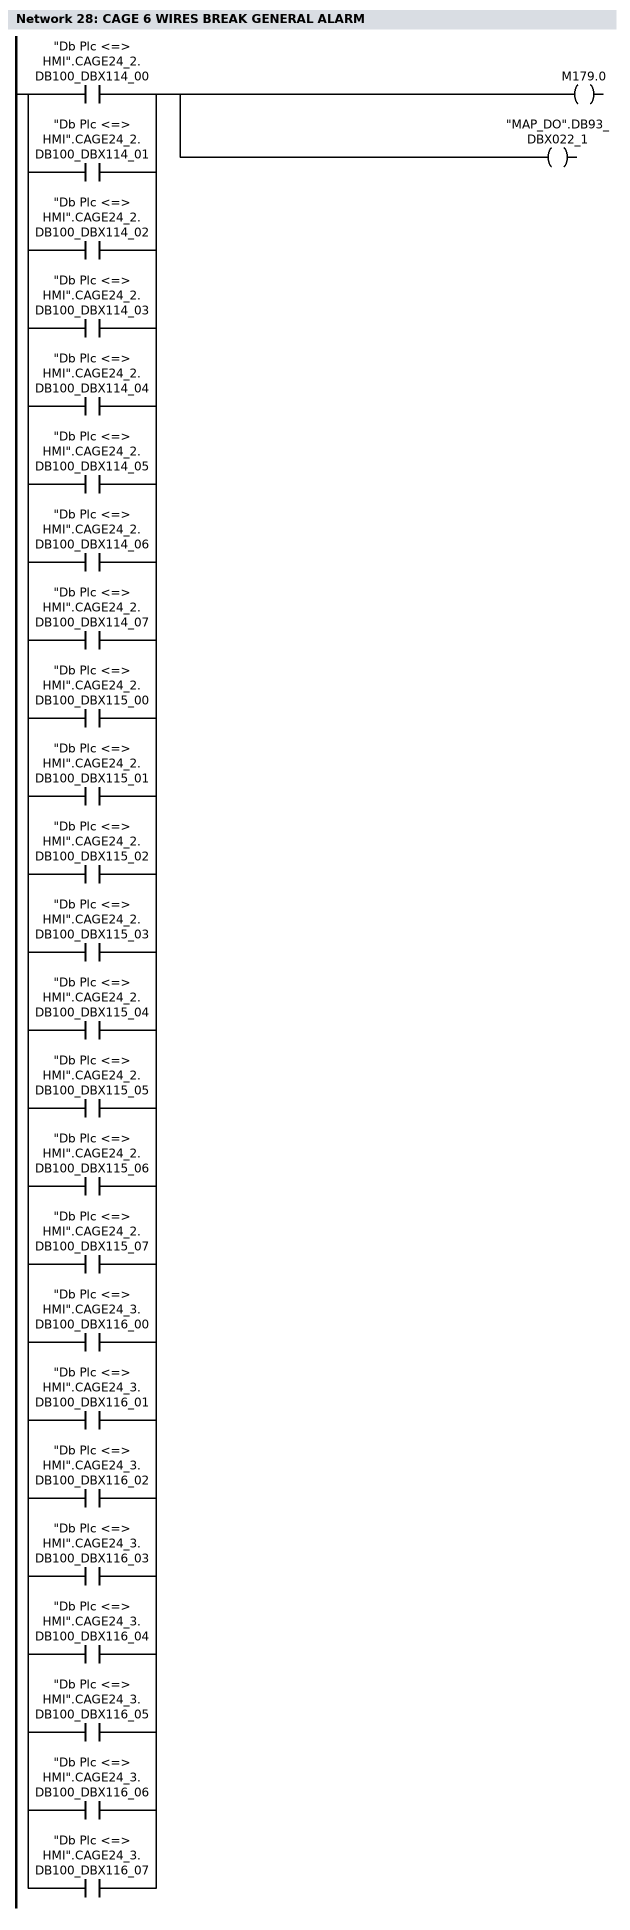
NETWORK
TITLE = CAGE 6 WIRES BREAK GENERAL ALARM
      O     "Db Plc <=> HMI".CAGE24_2.DB100_DBX114_00;
      O     "Db Plc <=> HMI".CAGE24_2.DB100_DBX114_01;
      O     "Db Plc <=> HMI".CAGE24_2.DB100_DBX114_02;
      O     "Db Plc <=> HMI".CAGE24_2.DB100_DBX114_03;
      O     "Db Plc <=> HMI".CAGE24_2.DB100_DBX114_04;
      O     "Db Plc <=> HMI".CAGE24_2.DB100_DBX114_05;
      O     "Db Plc <=> HMI".CAGE24_2.DB100_DBX114_06;
      O     "Db Plc <=> HMI".CAGE24_2.DB100_DBX114_07;
      O     "Db Plc <=> HMI".CAGE24_2.DB100_DBX115_00;
      O     "Db Plc <=> HMI".CAGE24_2.DB100_DBX115_01;
      O     "Db Plc <=> HMI".CAGE24_2.DB100_DBX115_02;
      O     "Db Plc <=> HMI".CAGE24_2.DB100_DBX115_03;
      O     "Db Plc <=> HMI".CAGE24_2.DB100_DBX115_04;
      O     "Db Plc <=> HMI".CAGE24_2.DB100_DBX115_05;
      O     "Db Plc <=> HMI".CAGE24_2.DB100_DBX115_06;
      O     "Db Plc <=> HMI".CAGE24_2.DB100_DBX115_07;
      O     "Db Plc <=> HMI".CAGE24_3.DB100_DBX116_00;
      O     "Db Plc <=> HMI".CAGE24_3.DB100_DBX116_01;
      O     "Db Plc <=> HMI".CAGE24_3.DB100_DBX116_02;
      O     "Db Plc <=> HMI".CAGE24_3.DB100_DBX116_03;
      O     "Db Plc <=> HMI".CAGE24_3.DB100_DBX116_04;
      O     "Db Plc <=> HMI".CAGE24_3.DB100_DBX116_05;
      O     "Db Plc <=> HMI".CAGE24_3.DB100_DBX116_06;
      O     "Db Plc <=> HMI".CAGE24_3.DB100_DBX116_07;
      =     "M179.0";
      =     "MAP_DO".DB93_DBX022_1;
END_FUNCTION

FUNCTION "Cage 18 wires insertion" : VOID	// FC 71
TITLE = CAGE 18 WIRES INSERTION AND ALARM FUNCTION
AUTHOR : Milesi
VERSION : 0.1
VAR_TEMP
  Tres : BOOL ;
END_VAR
BEGIN
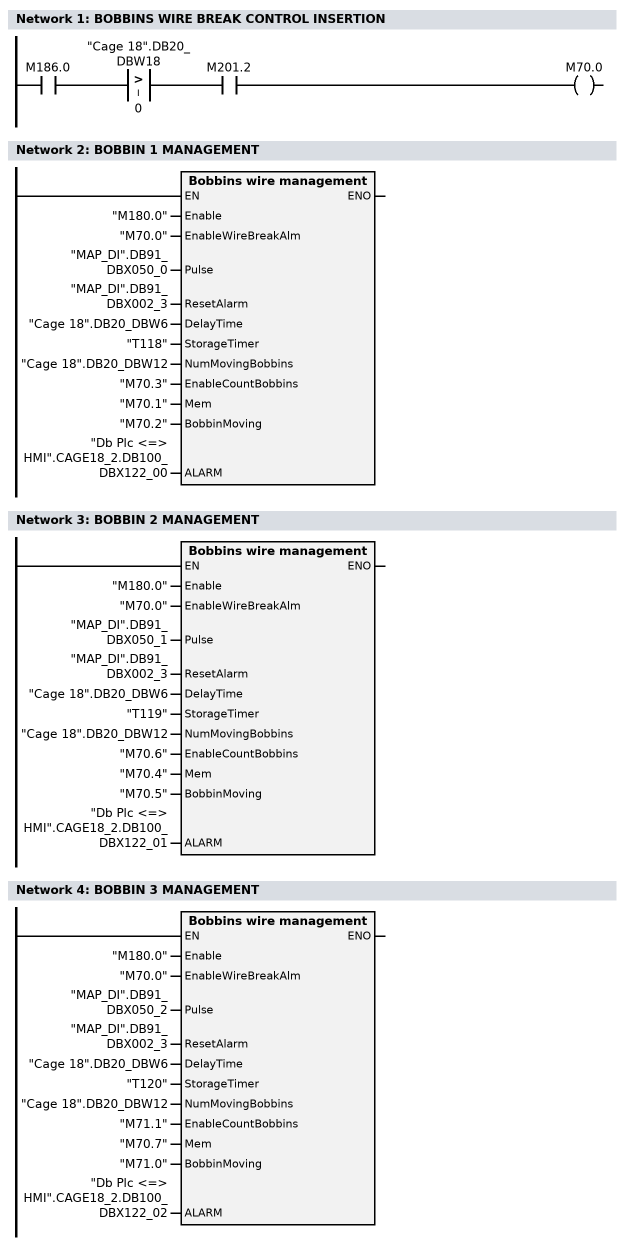
NETWORK
TITLE = BOBBINS WIRE BREAK CONTROL INSERTION
      A     "M186.0";
      A(;
      L     "Cage 18".DB20_DBW18;
      L     0;
      >I;
      );
      A     "M201.2";
      =     "M70.0";
NETWORK
TITLE = BOBBIN 1 MANAGEMENT
      CALL  "Bobbins wire management" (
           Enable                   := "M180.0",
           EnableWireBreakAlm       := "M70.0",
           Pulse                    := "MAP_DI".DB91_DBX050_0,
           ResetAlarm               := "MAP_DI".DB91_DBX002_3,
           DelayTime                := "Cage 18".DB20_DBW6,
           StorageTimer             := "T118",
           NumMovingBobbins         := "Cage 18".DB20_DBW12,
           EnableCountBobbins       := "M70.3",
           Mem                      := "M70.1",
           BobbinMoving             := "M70.2",
           ALARM                    := "Db Plc <=> HMI".CAGE18_2.DB100_DBX122_00);
      NOP   0;
NETWORK
TITLE = BOBBIN 2 MANAGEMENT
      CALL  "Bobbins wire management" (
           Enable                   := "M180.0",
           EnableWireBreakAlm       := "M70.0",
           Pulse                    := "MAP_DI".DB91_DBX050_1,
           ResetAlarm               := "MAP_DI".DB91_DBX002_3,
           DelayTime                := "Cage 18".DB20_DBW6,
           StorageTimer             := "T119",
           NumMovingBobbins         := "Cage 18".DB20_DBW12,
           EnableCountBobbins       := "M70.6",
           Mem                      := "M70.4",
           BobbinMoving             := "M70.5",
           ALARM                    := "Db Plc <=> HMI".CAGE18_2.DB100_DBX122_01);
NETWORK
TITLE = BOBBIN 3 MANAGEMENT
      CALL  "Bobbins wire management" (
           Enable                   := "M180.0",
           EnableWireBreakAlm       := "M70.0",
           Pulse                    := "MAP_DI".DB91_DBX050_2,
           ResetAlarm               := "MAP_DI".DB91_DBX002_3,
           DelayTime                := "Cage 18".DB20_DBW6,
           StorageTimer             := "T120",
           NumMovingBobbins         := "Cage 18".DB20_DBW12,
           EnableCountBobbins       := "M71.1",
           Mem                      := "M70.7",
           BobbinMoving             := "M71.0",
           ALARM                    := "Db Plc <=> HMI".CAGE18_2.DB100_DBX122_02);
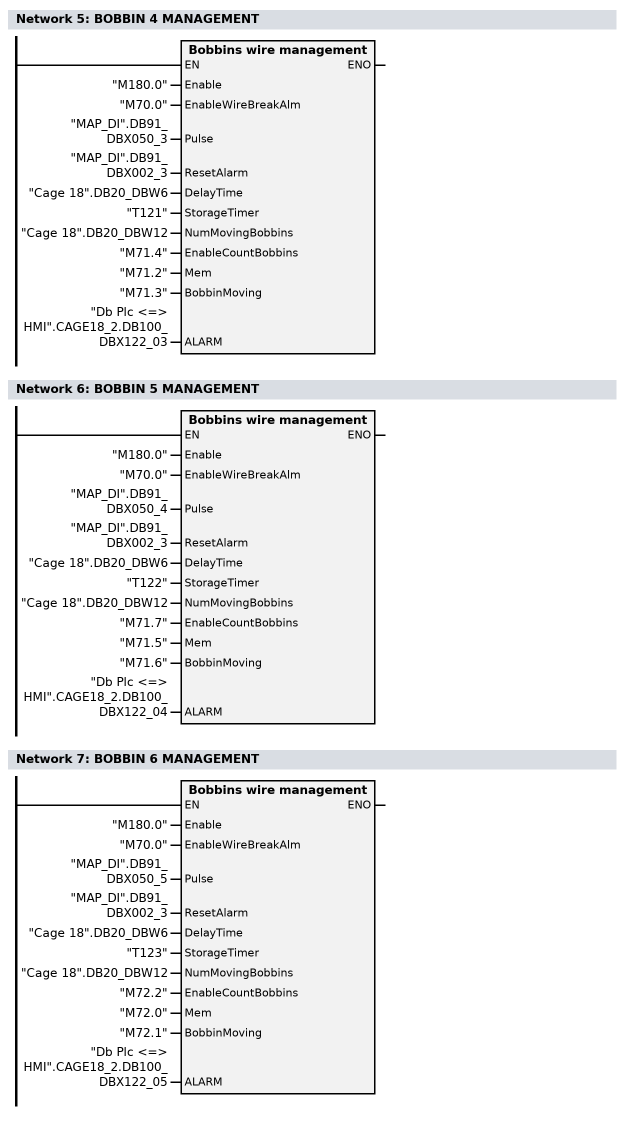
NETWORK
TITLE = BOBBIN 4 MANAGEMENT
      CALL  "Bobbins wire management" (
           Enable                   := "M180.0",
           EnableWireBreakAlm       := "M70.0",
           Pulse                    := "MAP_DI".DB91_DBX050_3,
           ResetAlarm               := "MAP_DI".DB91_DBX002_3,
           DelayTime                := "Cage 18".DB20_DBW6,
           StorageTimer             := "T121",
           NumMovingBobbins         := "Cage 18".DB20_DBW12,
           EnableCountBobbins       := "M71.4",
           Mem                      := "M71.2",
           BobbinMoving             := "M71.3",
           ALARM                    := "Db Plc <=> HMI".CAGE18_2.DB100_DBX122_03);
NETWORK
TITLE = BOBBIN 5 MANAGEMENT
      CALL  "Bobbins wire management" (
           Enable                   := "M180.0",
           EnableWireBreakAlm       := "M70.0",
           Pulse                    := "MAP_DI".DB91_DBX050_4,
           ResetAlarm               := "MAP_DI".DB91_DBX002_3,
           DelayTime                := "Cage 18".DB20_DBW6,
           StorageTimer             := "T122",
           NumMovingBobbins         := "Cage 18".DB20_DBW12,
           EnableCountBobbins       := "M71.7",
           Mem                      := "M71.5",
           BobbinMoving             := "M71.6",
           ALARM                    := "Db Plc <=> HMI".CAGE18_2.DB100_DBX122_04);
NETWORK
TITLE = BOBBIN 6 MANAGEMENT
      CALL  "Bobbins wire management" (
           Enable                   := "M180.0",
           EnableWireBreakAlm       := "M70.0",
           Pulse                    := "MAP_DI".DB91_DBX050_5,
           ResetAlarm               := "MAP_DI".DB91_DBX002_3,
           DelayTime                := "Cage 18".DB20_DBW6,
           StorageTimer             := "T123",
           NumMovingBobbins         := "Cage 18".DB20_DBW12,
           EnableCountBobbins       := "M72.2",
           Mem                      := "M72.0",
           BobbinMoving             := "M72.1",
           ALARM                    := "Db Plc <=> HMI".CAGE18_2.DB100_DBX122_05);
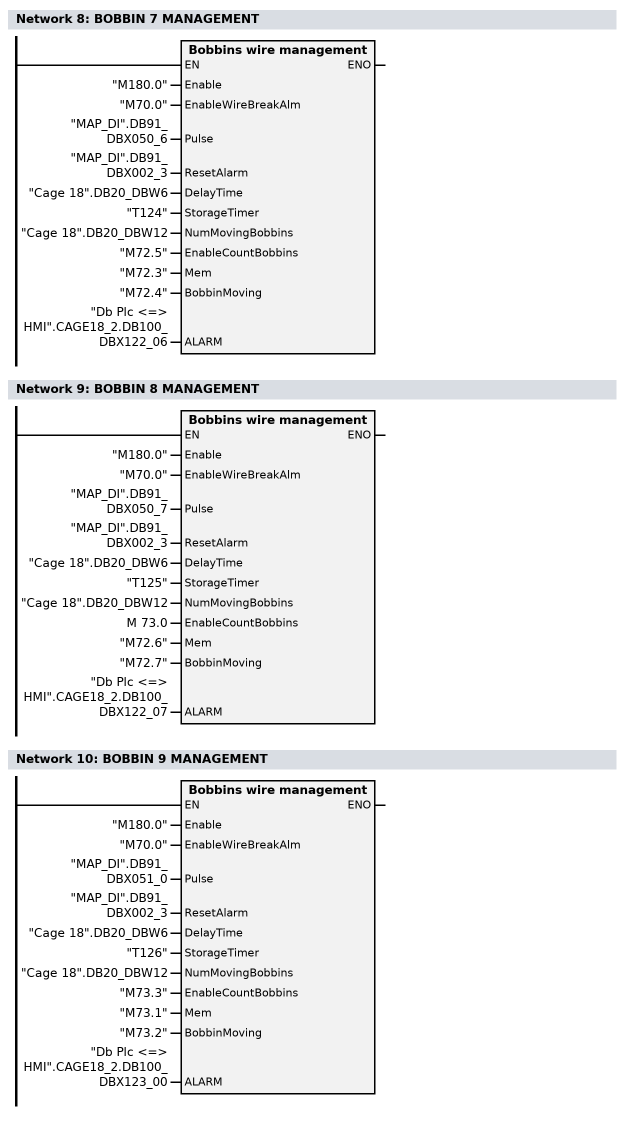
NETWORK
TITLE = BOBBIN 7 MANAGEMENT
      CALL  "Bobbins wire management" (
           Enable                   := "M180.0",
           EnableWireBreakAlm       := "M70.0",
           Pulse                    := "MAP_DI".DB91_DBX050_6,
           ResetAlarm               := "MAP_DI".DB91_DBX002_3,
           DelayTime                := "Cage 18".DB20_DBW6,
           StorageTimer             := "T124",
           NumMovingBobbins         := "Cage 18".DB20_DBW12,
           EnableCountBobbins       := "M72.5",
           Mem                      := "M72.3",
           BobbinMoving             := "M72.4",
           ALARM                    := "Db Plc <=> HMI".CAGE18_2.DB100_DBX122_06);
NETWORK
TITLE = BOBBIN 8 MANAGEMENT
      CALL  "Bobbins wire management" (
           Enable                   := "M180.0",
           EnableWireBreakAlm       := "M70.0",
           Pulse                    := "MAP_DI".DB91_DBX050_7,
           ResetAlarm               := "MAP_DI".DB91_DBX002_3,
           DelayTime                := "Cage 18".DB20_DBW6,
           StorageTimer             := "T125",
           NumMovingBobbins         := "Cage 18".DB20_DBW12,
           EnableCountBobbins       := M 73.0,
           Mem                      := "M72.6",
           BobbinMoving             := "M72.7",
           ALARM                    := "Db Plc <=> HMI".CAGE18_2.DB100_DBX122_07);
NETWORK
TITLE = BOBBIN 9 MANAGEMENT
      CALL  "Bobbins wire management" (
           Enable                   := "M180.0",
           EnableWireBreakAlm       := "M70.0",
           Pulse                    := "MAP_DI".DB91_DBX051_0,
           ResetAlarm               := "MAP_DI".DB91_DBX002_3,
           DelayTime                := "Cage 18".DB20_DBW6,
           StorageTimer             := "T126",
           NumMovingBobbins         := "Cage 18".DB20_DBW12,
           EnableCountBobbins       := "M73.3",
           Mem                      := "M73.1",
           BobbinMoving             := "M73.2",
           ALARM                    := "Db Plc <=> HMI".CAGE18_2.DB100_DBX123_00);
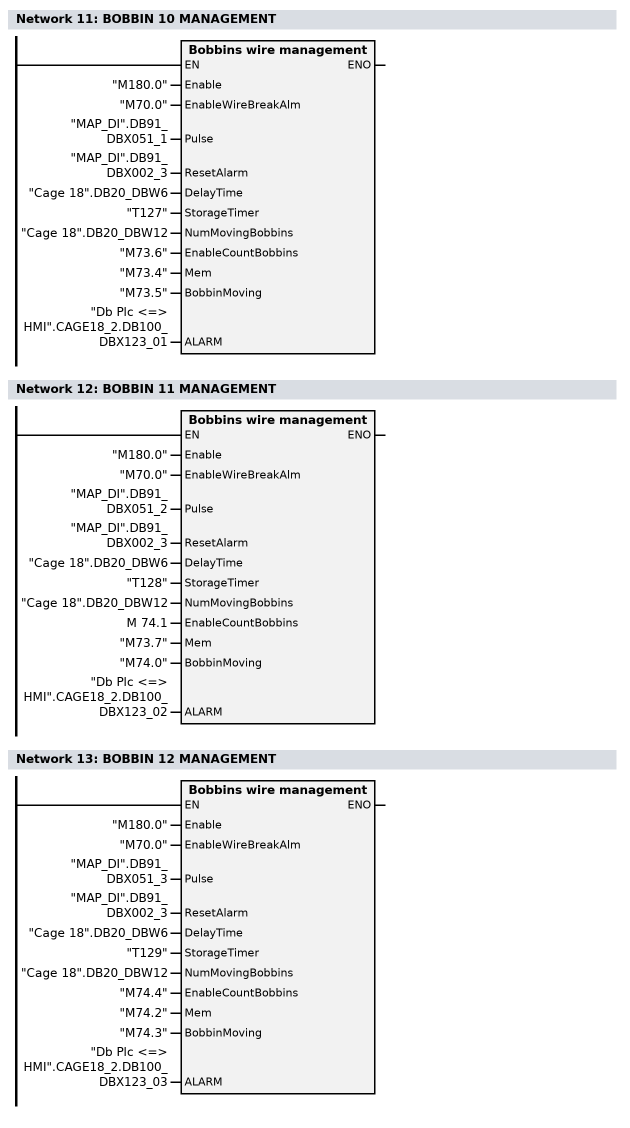
NETWORK
TITLE = BOBBIN 10 MANAGEMENT
      CALL  "Bobbins wire management" (
           Enable                   := "M180.0",
           EnableWireBreakAlm       := "M70.0",
           Pulse                    := "MAP_DI".DB91_DBX051_1,
           ResetAlarm               := "MAP_DI".DB91_DBX002_3,
           DelayTime                := "Cage 18".DB20_DBW6,
           StorageTimer             := "T127",
           NumMovingBobbins         := "Cage 18".DB20_DBW12,
           EnableCountBobbins       := "M73.6",
           Mem                      := "M73.4",
           BobbinMoving             := "M73.5",
           ALARM                    := "Db Plc <=> HMI".CAGE18_2.DB100_DBX123_01);
NETWORK
TITLE = BOBBIN 11 MANAGEMENT
      CALL  "Bobbins wire management" (
           Enable                   := "M180.0",
           EnableWireBreakAlm       := "M70.0",
           Pulse                    := "MAP_DI".DB91_DBX051_2,
           ResetAlarm               := "MAP_DI".DB91_DBX002_3,
           DelayTime                := "Cage 18".DB20_DBW6,
           StorageTimer             := "T128",
           NumMovingBobbins         := "Cage 18".DB20_DBW12,
           EnableCountBobbins       := M 74.1,
           Mem                      := "M73.7",
           BobbinMoving             := "M74.0",
           ALARM                    := "Db Plc <=> HMI".CAGE18_2.DB100_DBX123_02);
NETWORK
TITLE = BOBBIN 12 MANAGEMENT
      CALL  "Bobbins wire management" (
           Enable                   := "M180.0",
           EnableWireBreakAlm       := "M70.0",
           Pulse                    := "MAP_DI".DB91_DBX051_3,
           ResetAlarm               := "MAP_DI".DB91_DBX002_3,
           DelayTime                := "Cage 18".DB20_DBW6,
           StorageTimer             := "T129",
           NumMovingBobbins         := "Cage 18".DB20_DBW12,
           EnableCountBobbins       := "M74.4",
           Mem                      := "M74.2",
           BobbinMoving             := "M74.3",
           ALARM                    := "Db Plc <=> HMI".CAGE18_2.DB100_DBX123_03);
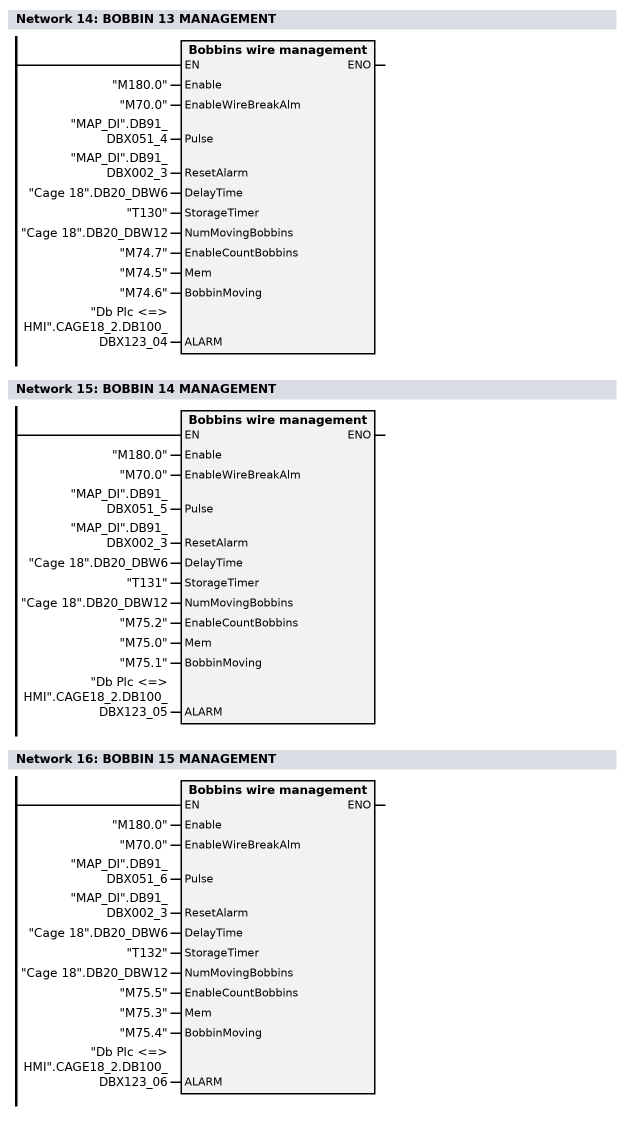
NETWORK
TITLE = BOBBIN 13 MANAGEMENT
      CALL  "Bobbins wire management" (
           Enable                   := "M180.0",
           EnableWireBreakAlm       := "M70.0",
           Pulse                    := "MAP_DI".DB91_DBX051_4,
           ResetAlarm               := "MAP_DI".DB91_DBX002_3,
           DelayTime                := "Cage 18".DB20_DBW6,
           StorageTimer             := "T130",
           NumMovingBobbins         := "Cage 18".DB20_DBW12,
           EnableCountBobbins       := "M74.7",
           Mem                      := "M74.5",
           BobbinMoving             := "M74.6",
           ALARM                    := "Db Plc <=> HMI".CAGE18_2.DB100_DBX123_04);
NETWORK
TITLE = BOBBIN 14 MANAGEMENT
      CALL  "Bobbins wire management" (
           Enable                   := "M180.0",
           EnableWireBreakAlm       := "M70.0",
           Pulse                    := "MAP_DI".DB91_DBX051_5,
           ResetAlarm               := "MAP_DI".DB91_DBX002_3,
           DelayTime                := "Cage 18".DB20_DBW6,
           StorageTimer             := "T131",
           NumMovingBobbins         := "Cage 18".DB20_DBW12,
           EnableCountBobbins       := "M75.2",
           Mem                      := "M75.0",
           BobbinMoving             := "M75.1",
           ALARM                    := "Db Plc <=> HMI".CAGE18_2.DB100_DBX123_05);
NETWORK
TITLE = BOBBIN 15 MANAGEMENT
      CALL  "Bobbins wire management" (
           Enable                   := "M180.0",
           EnableWireBreakAlm       := "M70.0",
           Pulse                    := "MAP_DI".DB91_DBX051_6,
           ResetAlarm               := "MAP_DI".DB91_DBX002_3,
           DelayTime                := "Cage 18".DB20_DBW6,
           StorageTimer             := "T132",
           NumMovingBobbins         := "Cage 18".DB20_DBW12,
           EnableCountBobbins       := "M75.5",
           Mem                      := "M75.3",
           BobbinMoving             := "M75.4",
           ALARM                    := "Db Plc <=> HMI".CAGE18_2.DB100_DBX123_06);
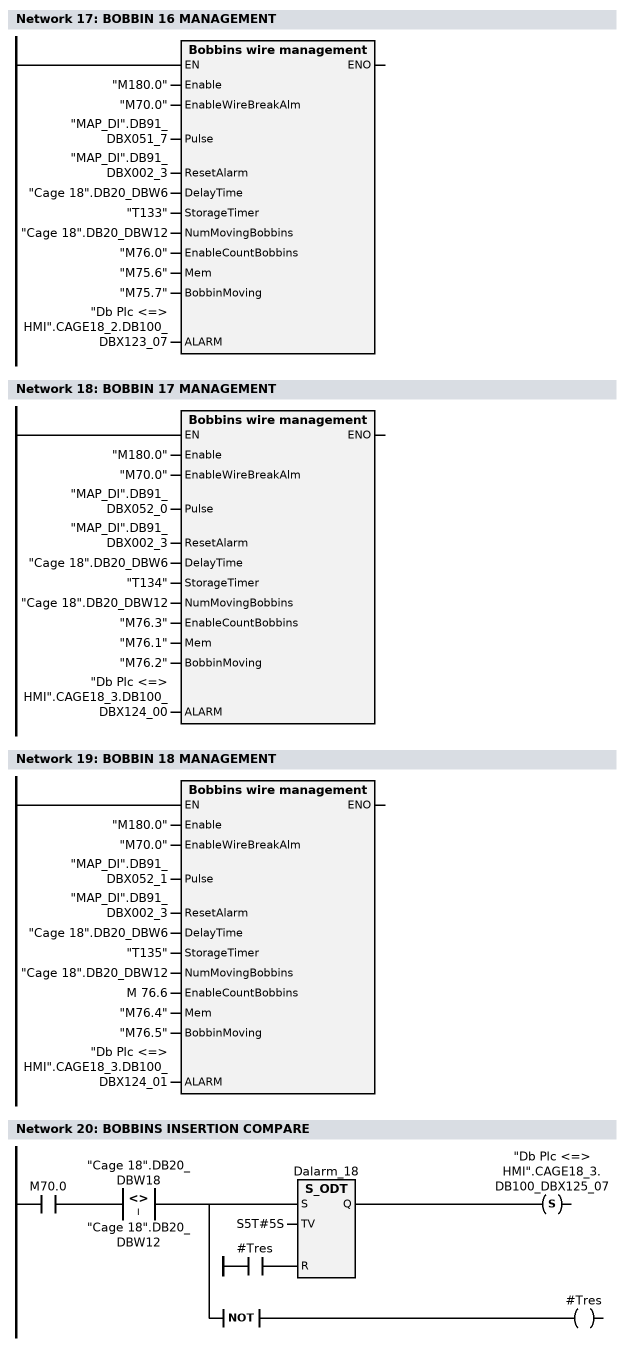
NETWORK
TITLE = BOBBIN 16 MANAGEMENT
      CALL  "Bobbins wire management" (
           Enable                   := "M180.0",
           EnableWireBreakAlm       := "M70.0",
           Pulse                    := "MAP_DI".DB91_DBX051_7,
           ResetAlarm               := "MAP_DI".DB91_DBX002_3,
           DelayTime                := "Cage 18".DB20_DBW6,
           StorageTimer             := "T133",
           NumMovingBobbins         := "Cage 18".DB20_DBW12,
           EnableCountBobbins       := "M76.0",
           Mem                      := "M75.6",
           BobbinMoving             := "M75.7",
           ALARM                    := "Db Plc <=> HMI".CAGE18_2.DB100_DBX123_07);
NETWORK
TITLE = BOBBIN 17 MANAGEMENT
      CALL  "Bobbins wire management" (
           Enable                   := "M180.0",
           EnableWireBreakAlm       := "M70.0",
           Pulse                    := "MAP_DI".DB91_DBX052_0,
           ResetAlarm               := "MAP_DI".DB91_DBX002_3,
           DelayTime                := "Cage 18".DB20_DBW6,
           StorageTimer             := "T134",
           NumMovingBobbins         := "Cage 18".DB20_DBW12,
           EnableCountBobbins       := "M76.3",
           Mem                      := "M76.1",
           BobbinMoving             := "M76.2",
           ALARM                    := "Db Plc <=> HMI".CAGE18_3.DB100_DBX124_00);
NETWORK
TITLE = BOBBIN 18 MANAGEMENT
      CALL  "Bobbins wire management" (
           Enable                   := "M180.0",
           EnableWireBreakAlm       := "M70.0",
           Pulse                    := "MAP_DI".DB91_DBX052_1,
           ResetAlarm               := "MAP_DI".DB91_DBX002_3,
           DelayTime                := "Cage 18".DB20_DBW6,
           StorageTimer             := "T135",
           NumMovingBobbins         := "Cage 18".DB20_DBW12,
           EnableCountBobbins       := M 76.6,
           Mem                      := "M76.4",
           BobbinMoving             := "M76.5",
           ALARM                    := "Db Plc <=> HMI".CAGE18_3.DB100_DBX124_01);
NETWORK
TITLE = BOBBINS INSERTION COMPARE
      A     "M70.0";
      A(;
      L     "Cage 18".DB20_DBW18;
      L     "Cage 18".DB20_DBW12;
      <>I;
      );
      =     L 1.0;
      A     L 1.0;
      L     S5T#5S;
      SD    "Dalarm_18";
      A     #Tres;
      R     "Dalarm_18";
      NOP   0;
      NOP   0;
      A     "Dalarm_18";
      S     "Db Plc <=> HMI".CAGE18_3.DB100_DBX125_07;
      A     L 1.0;
      NOT;
      =     #Tres;
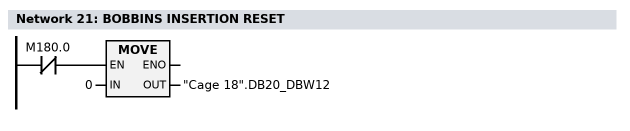
NETWORK
TITLE = BOBBINS INSERTION RESET
      AN    "M180.0";
      JNB   _001;
      L     0;
      T     "Cage 18".DB20_DBW12;
_001: NOP   0;
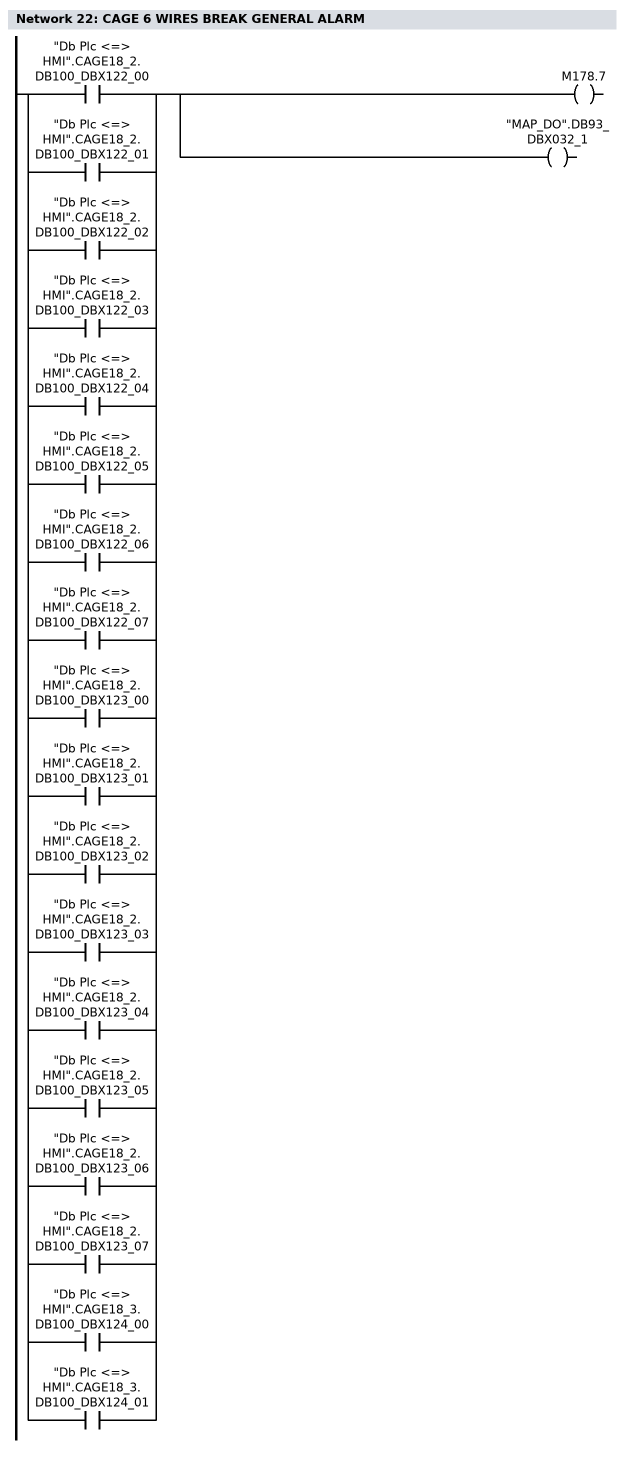
NETWORK
TITLE = CAGE 6 WIRES BREAK GENERAL ALARM
      O     "Db Plc <=> HMI".CAGE18_2.DB100_DBX122_00;
      O     "Db Plc <=> HMI".CAGE18_2.DB100_DBX122_01;
      O     "Db Plc <=> HMI".CAGE18_2.DB100_DBX122_02;
      O     "Db Plc <=> HMI".CAGE18_2.DB100_DBX122_03;
      O     "Db Plc <=> HMI".CAGE18_2.DB100_DBX122_04;
      O     "Db Plc <=> HMI".CAGE18_2.DB100_DBX122_05;
      O     "Db Plc <=> HMI".CAGE18_2.DB100_DBX122_06;
      O     "Db Plc <=> HMI".CAGE18_2.DB100_DBX122_07;
      O     "Db Plc <=> HMI".CAGE18_2.DB100_DBX123_00;
      O     "Db Plc <=> HMI".CAGE18_2.DB100_DBX123_01;
      O     "Db Plc <=> HMI".CAGE18_2.DB100_DBX123_02;
      O     "Db Plc <=> HMI".CAGE18_2.DB100_DBX123_03;
      O     "Db Plc <=> HMI".CAGE18_2.DB100_DBX123_04;
      O     "Db Plc <=> HMI".CAGE18_2.DB100_DBX123_05;
      O     "Db Plc <=> HMI".CAGE18_2.DB100_DBX123_06;
      O     "Db Plc <=> HMI".CAGE18_2.DB100_DBX123_07;
      O     "Db Plc <=> HMI".CAGE18_3.DB100_DBX124_00;
      O     "Db Plc <=> HMI".CAGE18_3.DB100_DBX124_01;
      =     "M178.7";
      =     "MAP_DO".DB93_DBX032_1;
END_FUNCTION

FUNCTION "Cage 12 wires insertion" : VOID	// FC 72
TITLE = CAGE 12 WIRES INSERTION AND ALARM FUNCTION
AUTHOR : Milesi
VERSION : 0.1
VAR_TEMP
  Tres : BOOL ;
END_VAR
BEGIN
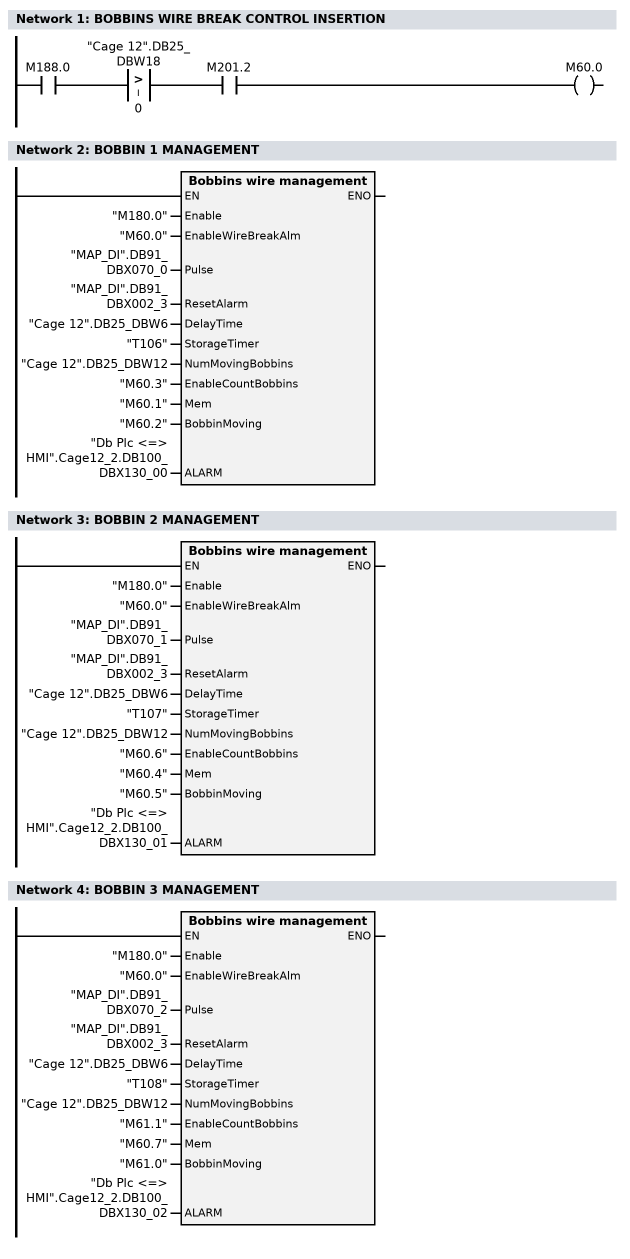
NETWORK
TITLE = BOBBINS WIRE BREAK CONTROL INSERTION
      A     "M188.0";
      A(;
      L     "Cage 12".DB25_DBW18;
      L     0;
      >I;
      );
      A     "M201.2";
      =     "M60.0";
NETWORK
TITLE = BOBBIN 1 MANAGEMENT
      CALL  "Bobbins wire management" (
           Enable                   := "M180.0",
           EnableWireBreakAlm       := "M60.0",
           Pulse                    := "MAP_DI".DB91_DBX070_0,
           ResetAlarm               := "MAP_DI".DB91_DBX002_3,
           DelayTime                := "Cage 12".DB25_DBW6,
           StorageTimer             := "T106",
           NumMovingBobbins         := "Cage 12".DB25_DBW12,
           EnableCountBobbins       := "M60.3",
           Mem                      := "M60.1",
           BobbinMoving             := "M60.2",
           ALARM                    := "Db Plc <=> HMI".Cage12_2.DB100_DBX130_00);
      NOP   0;
NETWORK
TITLE = BOBBIN 2 MANAGEMENT
      CALL  "Bobbins wire management" (
           Enable                   := "M180.0",
           EnableWireBreakAlm       := "M60.0",
           Pulse                    := "MAP_DI".DB91_DBX070_1,
           ResetAlarm               := "MAP_DI".DB91_DBX002_3,
           DelayTime                := "Cage 12".DB25_DBW6,
           StorageTimer             := "T107",
           NumMovingBobbins         := "Cage 12".DB25_DBW12,
           EnableCountBobbins       := "M60.6",
           Mem                      := "M60.4",
           BobbinMoving             := "M60.5",
           ALARM                    := "Db Plc <=> HMI".Cage12_2.DB100_DBX130_01);
NETWORK
TITLE = BOBBIN 3 MANAGEMENT
      CALL  "Bobbins wire management" (
           Enable                   := "M180.0",
           EnableWireBreakAlm       := "M60.0",
           Pulse                    := "MAP_DI".DB91_DBX070_2,
           ResetAlarm               := "MAP_DI".DB91_DBX002_3,
           DelayTime                := "Cage 12".DB25_DBW6,
           StorageTimer             := "T108",
           NumMovingBobbins         := "Cage 12".DB25_DBW12,
           EnableCountBobbins       := "M61.1",
           Mem                      := "M60.7",
           BobbinMoving             := "M61.0",
           ALARM                    := "Db Plc <=> HMI".Cage12_2.DB100_DBX130_02);
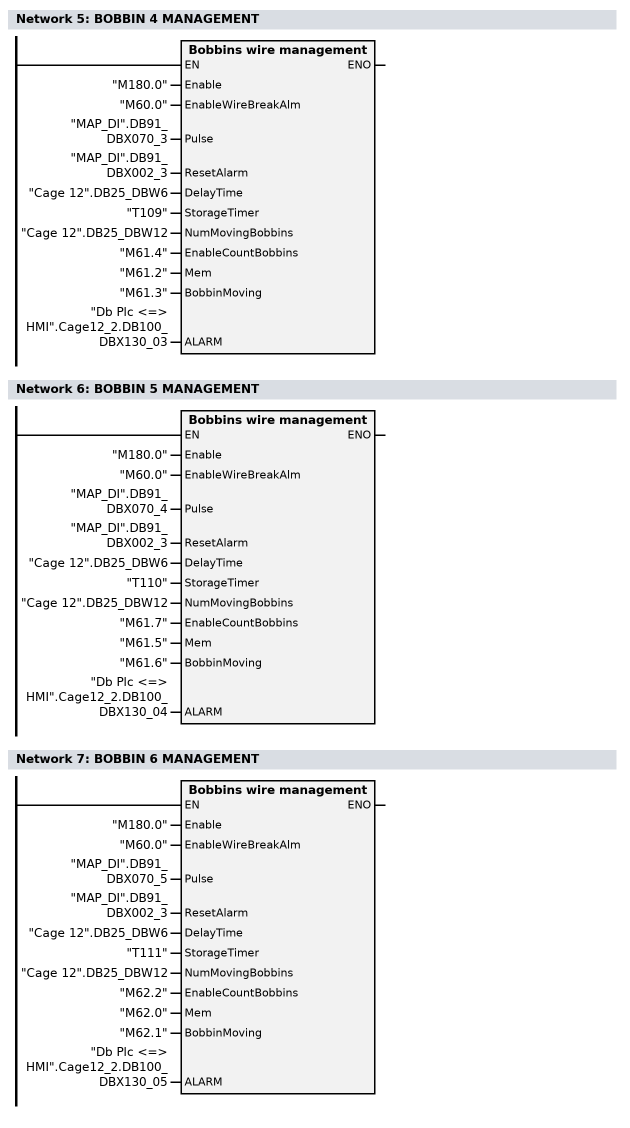
NETWORK
TITLE = BOBBIN 4 MANAGEMENT
      CALL  "Bobbins wire management" (
           Enable                   := "M180.0",
           EnableWireBreakAlm       := "M60.0",
           Pulse                    := "MAP_DI".DB91_DBX070_3,
           ResetAlarm               := "MAP_DI".DB91_DBX002_3,
           DelayTime                := "Cage 12".DB25_DBW6,
           StorageTimer             := "T109",
           NumMovingBobbins         := "Cage 12".DB25_DBW12,
           EnableCountBobbins       := "M61.4",
           Mem                      := "M61.2",
           BobbinMoving             := "M61.3",
           ALARM                    := "Db Plc <=> HMI".Cage12_2.DB100_DBX130_03);
NETWORK
TITLE = BOBBIN 5 MANAGEMENT
      CALL  "Bobbins wire management" (
           Enable                   := "M180.0",
           EnableWireBreakAlm       := "M60.0",
           Pulse                    := "MAP_DI".DB91_DBX070_4,
           ResetAlarm               := "MAP_DI".DB91_DBX002_3,
           DelayTime                := "Cage 12".DB25_DBW6,
           StorageTimer             := "T110",
           NumMovingBobbins         := "Cage 12".DB25_DBW12,
           EnableCountBobbins       := "M61.7",
           Mem                      := "M61.5",
           BobbinMoving             := "M61.6",
           ALARM                    := "Db Plc <=> HMI".Cage12_2.DB100_DBX130_04);
NETWORK
TITLE = BOBBIN 6 MANAGEMENT
      CALL  "Bobbins wire management" (
           Enable                   := "M180.0",
           EnableWireBreakAlm       := "M60.0",
           Pulse                    := "MAP_DI".DB91_DBX070_5,
           ResetAlarm               := "MAP_DI".DB91_DBX002_3,
           DelayTime                := "Cage 12".DB25_DBW6,
           StorageTimer             := "T111",
           NumMovingBobbins         := "Cage 12".DB25_DBW12,
           EnableCountBobbins       := "M62.2",
           Mem                      := "M62.0",
           BobbinMoving             := "M62.1",
           ALARM                    := "Db Plc <=> HMI".Cage12_2.DB100_DBX130_05);
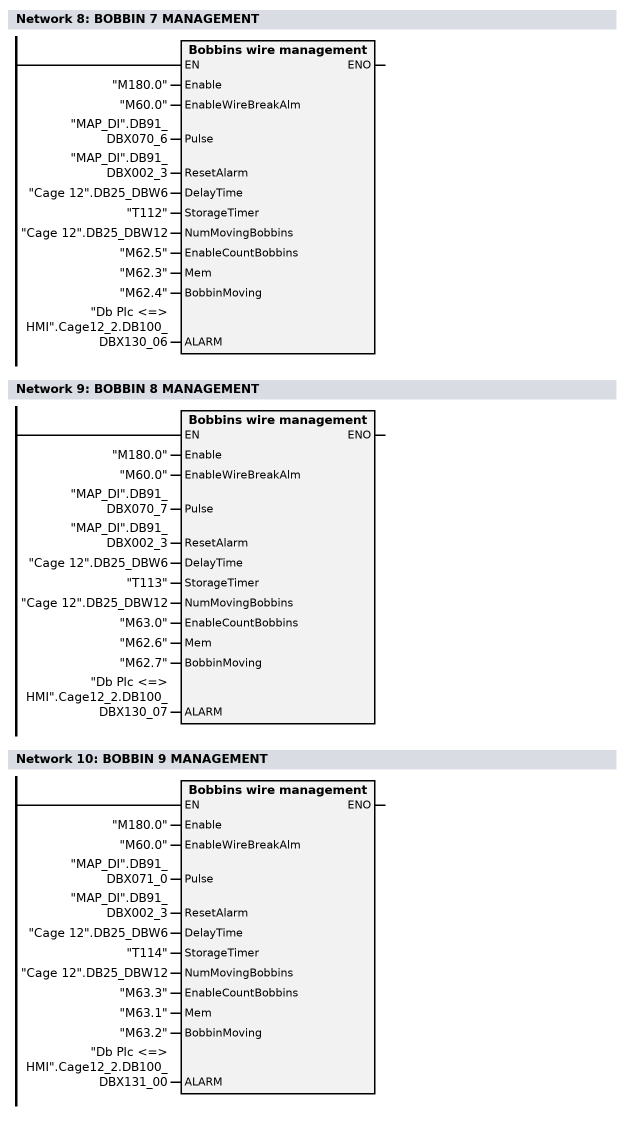
NETWORK
TITLE = BOBBIN 7 MANAGEMENT
      CALL  "Bobbins wire management" (
           Enable                   := "M180.0",
           EnableWireBreakAlm       := "M60.0",
           Pulse                    := "MAP_DI".DB91_DBX070_6,
           ResetAlarm               := "MAP_DI".DB91_DBX002_3,
           DelayTime                := "Cage 12".DB25_DBW6,
           StorageTimer             := "T112",
           NumMovingBobbins         := "Cage 12".DB25_DBW12,
           EnableCountBobbins       := "M62.5",
           Mem                      := "M62.3",
           BobbinMoving             := "M62.4",
           ALARM                    := "Db Plc <=> HMI".Cage12_2.DB100_DBX130_06);
NETWORK
TITLE = BOBBIN 8 MANAGEMENT
      CALL  "Bobbins wire management" (
           Enable                   := "M180.0",
           EnableWireBreakAlm       := "M60.0",
           Pulse                    := "MAP_DI".DB91_DBX070_7,
           ResetAlarm               := "MAP_DI".DB91_DBX002_3,
           DelayTime                := "Cage 12".DB25_DBW6,
           StorageTimer             := "T113",
           NumMovingBobbins         := "Cage 12".DB25_DBW12,
           EnableCountBobbins       := "M63.0",
           Mem                      := "M62.6",
           BobbinMoving             := "M62.7",
           ALARM                    := "Db Plc <=> HMI".Cage12_2.DB100_DBX130_07);
NETWORK
TITLE = BOBBIN 9 MANAGEMENT
      CALL  "Bobbins wire management" (
           Enable                   := "M180.0",
           EnableWireBreakAlm       := "M60.0",
           Pulse                    := "MAP_DI".DB91_DBX071_0,
           ResetAlarm               := "MAP_DI".DB91_DBX002_3,
           DelayTime                := "Cage 12".DB25_DBW6,
           StorageTimer             := "T114",
           NumMovingBobbins         := "Cage 12".DB25_DBW12,
           EnableCountBobbins       := "M63.3",
           Mem                      := "M63.1",
           BobbinMoving             := "M63.2",
           ALARM                    := "Db Plc <=> HMI".Cage12_2.DB100_DBX131_00);
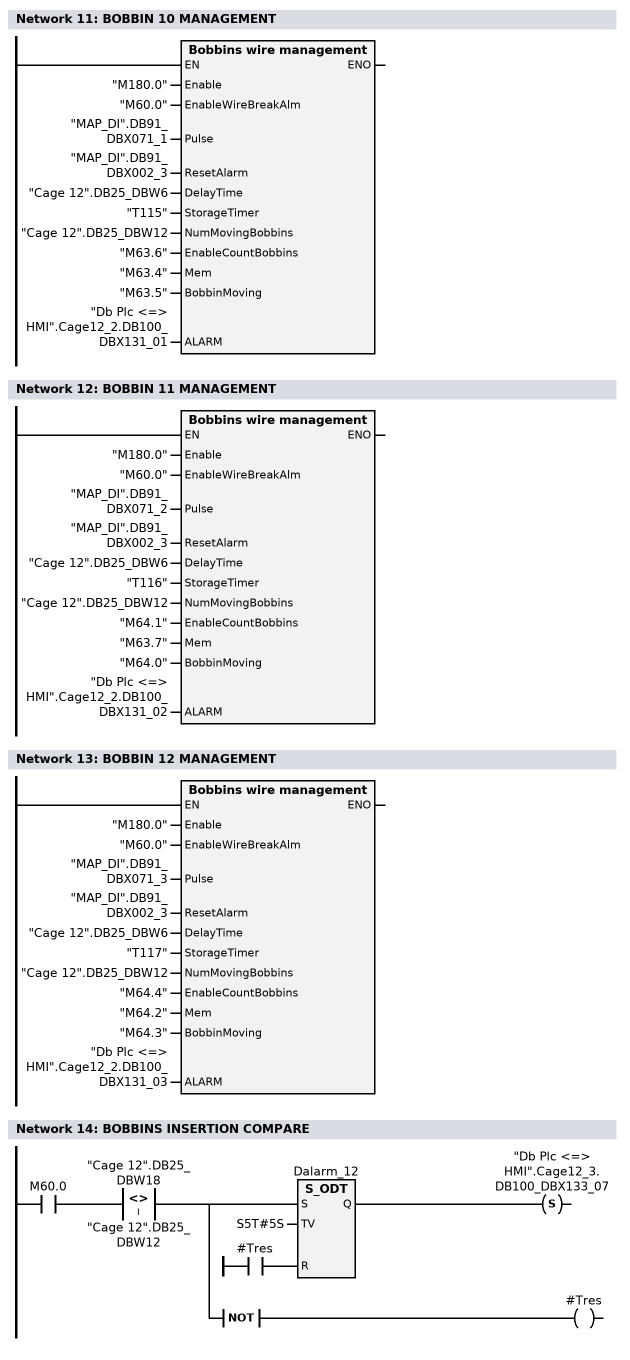
NETWORK
TITLE = BOBBIN 10 MANAGEMENT
      CALL  "Bobbins wire management" (
           Enable                   := "M180.0",
           EnableWireBreakAlm       := "M60.0",
           Pulse                    := "MAP_DI".DB91_DBX071_1,
           ResetAlarm               := "MAP_DI".DB91_DBX002_3,
           DelayTime                := "Cage 12".DB25_DBW6,
           StorageTimer             := "T115",
           NumMovingBobbins         := "Cage 12".DB25_DBW12,
           EnableCountBobbins       := "M63.6",
           Mem                      := "M63.4",
           BobbinMoving             := "M63.5",
           ALARM                    := "Db Plc <=> HMI".Cage12_2.DB100_DBX131_01);
NETWORK
TITLE = BOBBIN 11 MANAGEMENT
      CALL  "Bobbins wire management" (
           Enable                   := "M180.0",
           EnableWireBreakAlm       := "M60.0",
           Pulse                    := "MAP_DI".DB91_DBX071_2,
           ResetAlarm               := "MAP_DI".DB91_DBX002_3,
           DelayTime                := "Cage 12".DB25_DBW6,
           StorageTimer             := "T116",
           NumMovingBobbins         := "Cage 12".DB25_DBW12,
           EnableCountBobbins       := "M64.1",
           Mem                      := "M63.7",
           BobbinMoving             := "M64.0",
           ALARM                    := "Db Plc <=> HMI".Cage12_2.DB100_DBX131_02);
NETWORK
TITLE = BOBBIN 12 MANAGEMENT
      CALL  "Bobbins wire management" (
           Enable                   := "M180.0",
           EnableWireBreakAlm       := "M60.0",
           Pulse                    := "MAP_DI".DB91_DBX071_3,
           ResetAlarm               := "MAP_DI".DB91_DBX002_3,
           DelayTime                := "Cage 12".DB25_DBW6,
           StorageTimer             := "T117",
           NumMovingBobbins         := "Cage 12".DB25_DBW12,
           EnableCountBobbins       := "M64.4",
           Mem                      := "M64.2",
           BobbinMoving             := "M64.3",
           ALARM                    := "Db Plc <=> HMI".Cage12_2.DB100_DBX131_03);
NETWORK
TITLE = BOBBINS INSERTION COMPARE
      A     "M60.0";
      A(;
      L     "Cage 12".DB25_DBW18;
      L     "Cage 12".DB25_DBW12;
      <>I;
      );
      =     L 1.0;
      A     L 1.0;
      L     S5T#5S;
      SD    "Dalarm_12";
      A     #Tres;
      R     "Dalarm_12";
      NOP   0;
      NOP   0;
      A     "Dalarm_12";
      S     "Db Plc <=> HMI".Cage12_3.DB100_DBX133_07;
      A     L 1.0;
      NOT;
      =     #Tres;
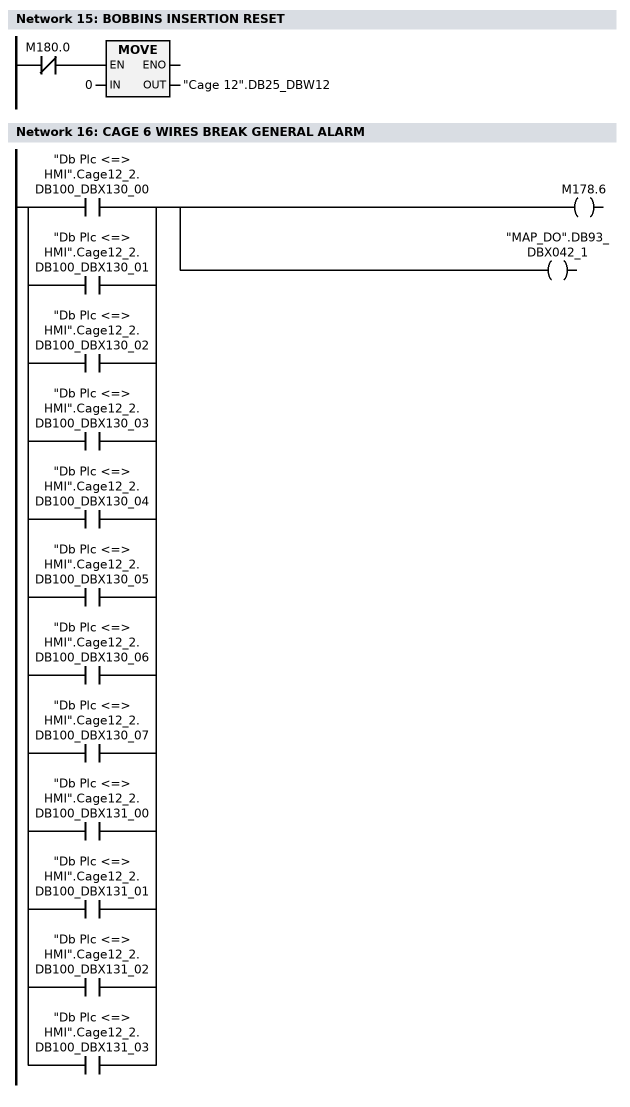
NETWORK
TITLE = BOBBINS INSERTION RESET
      AN    "M180.0";
      JNB   _001;
      L     0;
      T     "Cage 12".DB25_DBW12;
_001: NOP   0;
NETWORK
TITLE = CAGE 6 WIRES BREAK GENERAL ALARM
      O     "Db Plc <=> HMI".Cage12_2.DB100_DBX130_00;
      O     "Db Plc <=> HMI".Cage12_2.DB100_DBX130_01;
      O     "Db Plc <=> HMI".Cage12_2.DB100_DBX130_02;
      O     "Db Plc <=> HMI".Cage12_2.DB100_DBX130_03;
      O     "Db Plc <=> HMI".Cage12_2.DB100_DBX130_04;
      O     "Db Plc <=> HMI".Cage12_2.DB100_DBX130_05;
      O     "Db Plc <=> HMI".Cage12_2.DB100_DBX130_06;
      O     "Db Plc <=> HMI".Cage12_2.DB100_DBX130_07;
      O     "Db Plc <=> HMI".Cage12_2.DB100_DBX131_00;
      O     "Db Plc <=> HMI".Cage12_2.DB100_DBX131_01;
      O     "Db Plc <=> HMI".Cage12_2.DB100_DBX131_02;
      O     "Db Plc <=> HMI".Cage12_2.DB100_DBX131_03;
      =     "M178.6";
      =     "MAP_DO".DB93_DBX042_1;
END_FUNCTION

FUNCTION "Cage 6 wires insertion" : VOID	// FC 73
TITLE = CAGE 6 WIRES INSERTION FUNCTION
AUTHOR : Milesi
VERSION : 0.1
VAR_TEMP
  Tres : BOOL ;
END_VAR
BEGIN
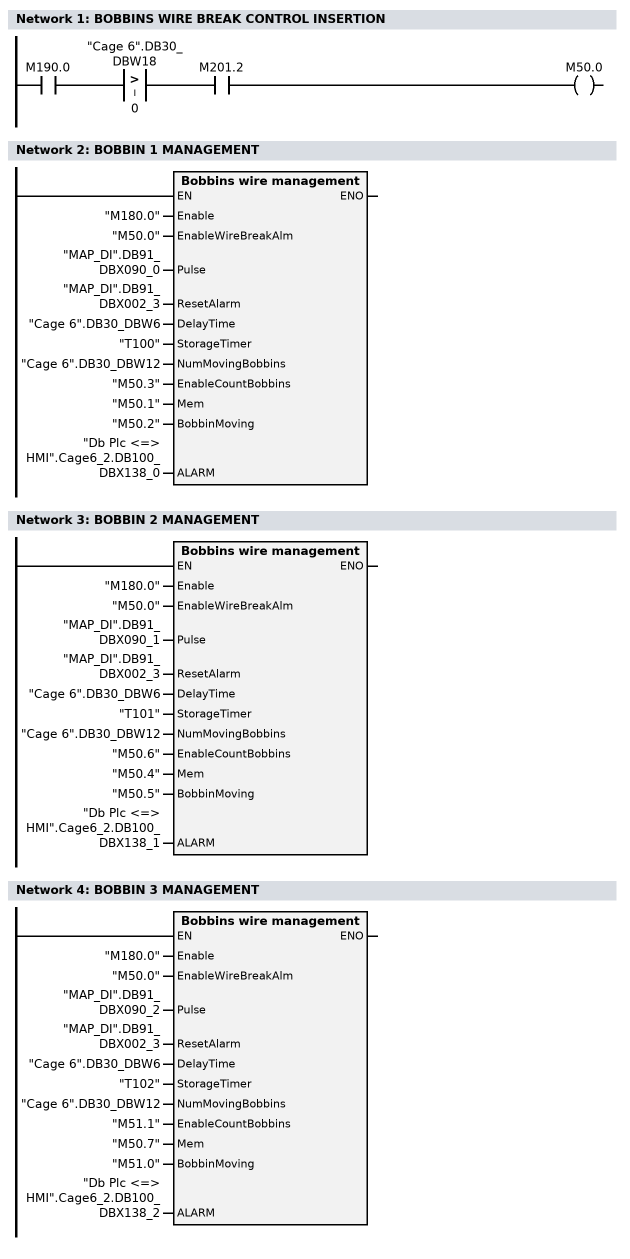
NETWORK
TITLE = BOBBINS WIRE BREAK CONTROL INSERTION
      A     "M190.0";
      A(;
      L     "Cage 6".DB30_DBW18;
      L     0;
      >I;
      );
      A     "M201.2";
      =     "M50.0";
NETWORK
TITLE = BOBBIN 1 MANAGEMENT
      CALL  "Bobbins wire management" (
           Enable                   := "M180.0",
           EnableWireBreakAlm       := "M50.0",
           Pulse                    := "MAP_DI".DB91_DBX090_0,
           ResetAlarm               := "MAP_DI".DB91_DBX002_3,
           DelayTime                := "Cage 6".DB30_DBW6,
           StorageTimer             := "T100",
           NumMovingBobbins         := "Cage 6".DB30_DBW12,
           EnableCountBobbins       := "M50.3",
           Mem                      := "M50.1",
           BobbinMoving             := "M50.2",
           ALARM                    := "Db Plc <=> HMI".Cage6_2.DB100_DBX138_0);
      NOP   0;
NETWORK
TITLE = BOBBIN 2 MANAGEMENT
      CALL  "Bobbins wire management" (
           Enable                   := "M180.0",
           EnableWireBreakAlm       := "M50.0",
           Pulse                    := "MAP_DI".DB91_DBX090_1,
           ResetAlarm               := "MAP_DI".DB91_DBX002_3,
           DelayTime                := "Cage 6".DB30_DBW6,
           StorageTimer             := "T101",
           NumMovingBobbins         := "Cage 6".DB30_DBW12,
           EnableCountBobbins       := "M50.6",
           Mem                      := "M50.4",
           BobbinMoving             := "M50.5",
           ALARM                    := "Db Plc <=> HMI".Cage6_2.DB100_DBX138_1);
NETWORK
TITLE = BOBBIN 3 MANAGEMENT
      CALL  "Bobbins wire management" (
           Enable                   := "M180.0",
           EnableWireBreakAlm       := "M50.0",
           Pulse                    := "MAP_DI".DB91_DBX090_2,
           ResetAlarm               := "MAP_DI".DB91_DBX002_3,
           DelayTime                := "Cage 6".DB30_DBW6,
           StorageTimer             := "T102",
           NumMovingBobbins         := "Cage 6".DB30_DBW12,
           EnableCountBobbins       := "M51.1",
           Mem                      := "M50.7",
           BobbinMoving             := "M51.0",
           ALARM                    := "Db Plc <=> HMI".Cage6_2.DB100_DBX138_2);
